// TIA Portal V20 export
FUNCTION_BLOCK "LER_Heater"   // FB21, LAD
// stored: Access Published, MemoryReserve 100, SetENOAutomatically false
   VAR_INPUT
      enable { ExternalAccessible := 'False'; ExternalVisible := 'False'; ExternalWritable := 'False'} : Bool;   // TRUE: Enable functionality of FB
      enableManualCmds : Bool;   // Enabling manual commands
      Clock : Bool;
   END_VAR
   VAR_OUTPUT
      Error : Bool;
   END_VAR
   VAR_IN_OUT
      ModbusMasterDataPTR : Variant;
      configuration : "LER_typeHeaterConfiguration";
      controlNode : "LER_typeHeaterControlNode";
      moduleInterface : "LER_typeHeaterInterface";
   END_VAR
   VAR
      statEnable : Bool;
      statEnableManualCmds : Bool;
      statSaveBtn : Bool;
      staSaveOneCycleDONE : Bool;
      instModbusCommLoad : Modbus_Comm_Load;
      instModbusMaster : Modbus_Master;
      instLER_Heater : Array[1.."Number_Of_E5CC"] of "LER_E5CC";
      "statE5CC[1]" { S7_SetPoint := 'True'} : "LER_typeE5CCStatus";
      "statE5CC[2]" { S7_SetPoint := 'True'} : "LER_typeE5CCStatus";
      "statE5CC[3]" { S7_SetPoint := 'True'} : "LER_typeE5CCStatus";
      "statE5CC[4]" { S7_SetPoint := 'True'} : "LER_typeE5CCStatus";
      "statE5CC[5]" { S7_SetPoint := 'True'} : "LER_typeE5CCStatus";
      statMBMasterBuffer { S7_SetPoint := 'True'} : Array[1.."Number_Of_E5CC"] of "LER_typeHeaterConfiguration_MB_Master";
      statCommand : "LER_typeHeaterCommands";
      statCMDKeep : Struct
         "E5CC[1]" : Struct
            Upper_Heater_Run : Bool;
            Upper_Heater_Stop : Bool;
            Upper_AutoTune_Run : Bool;
            Upper_AutoTune_Stop : Bool;
         END_STRUCT;
         "E5CC[2]" : Struct
            Upper_Heater_Run : Bool;
            Upper_Heater_Stop : Bool;
            Upper_AutoTune_Run : Bool;
            Upper_AutoTune_Stop : Bool;
         END_STRUCT;
         "E5CC[3]" : Struct
            Upper_Heater_Run : Bool;
            Upper_Heater_Stop : Bool;
            Upper_AutoTune_Run : Bool;
            Upper_AutoTune_Stop : Bool;
         END_STRUCT;
         "E5CC[4]" : Struct
            Upper_Heater_Run : Bool;
            Upper_Heater_Stop : Bool;
            Upper_AutoTune_Run : Bool;
            Upper_AutoTune_Stop : Bool;
         END_STRUCT;
         "E5CC[5]" : Struct
            Upper_Heater_Run : Bool;
            Upper_Heater_Stop : Bool;
            Upper_AutoTune_Run : Bool;
            Upper_AutoTune_Stop : Bool;
         END_STRUCT;
         E5CC1ReadStop : Bool;
         E5CC2ReadStop : Bool;
         E5CC3ReadStop : Bool;
         E5CC4ReadStop : Bool;
         E5CC5ReadStop : Bool;
      END_STRUCT;
      statConfiguration : "LER_typeHeaterConfiguration";
      statMonitoring { S7_SetPoint := 'True'} : "LER_typeHeaterMonitoring";
      statCurrentUnit : Int := 1;
      statTimer : Array[0..30] of TON_TIME;
      statPulse : Array[0..59] of Bool;
      IEC_Timer_0_Instance { S7_SetPoint := 'True'} : TOF_TIME;
      IEC_Timer_0_Instance_1 { S7_SetPoint := 'True'} : TOF_TIME;
      IEC_Timer_0_Instance_2 { S7_SetPoint := 'True'} : TOF_TIME;
      IEC_Timer_0_Instance_3 { S7_SetPoint := 'True'} : TOF_TIME;
      IEC_Timer_0_Instance_4 { S7_SetPoint := 'True'} : TOF_TIME;
   END_VAR
   VAR_TEMP
      tempErrInt : Int;
      tempErrWord : Word;
   END_VAR
   VAR CONSTANT
      Addr_TempPV : UDInt := 40001;
      Addr_Status : UDInt := 40003;
      Addr_TempSP : UDInt := 40263;
      Addr_AlarmValue1 : UDInt := 40265;
      Addr_AlarmValue1_UpperLimit : UDInt := 40267;
      Addr_AlarmValue1_LowerLimit : UDInt := 40269;
      Addr_AlarmValue2 : UDInt := 40271;
      Addr_AlarmValue2_UpperLimit : UDInt := 40273;
      Addr_AlarmValue2_LowerLimit : UDInt := 40275;
      CMD_Run : DWord := 16#01000000;
      CMD_Stop : DWord := 16#01010000;
      CMD_AutoTune_Run : DWord := 16#03020000;
      CMD_AutoTune_Stop : DWord := 16#03000000;
      Mode_Read : Int := 0;
      Mode_Write : Int := 1;
      Read_Time : Time := T#500MS;
      STATUS_NO_ERROR_OCCURRED : DWord;   // No error occurred.
      ERR_HEATER_CURRENT_VALUE_EXCEEDED_CT1 : DWord := 16#1;
      ERR_HEATER_CURRENT_VALUE_HOLD_CT1 : DWord := 16#2;
      ERR_AD_CONVERTER_ABNORMALITY : DWord := 16#4;
      ERR_HS_SSR_FAULT_ALERT_CT1 : DWord := 16#8;
      ERR_RSP_INPUT_ABNORMALITIES : DWord := 16#10;
      ERR_MORE_THAN_INPUT : DWord := 16#40;
      ERR_POTENTIOMETER_INPUT_ABNORMAL : DWord := 16#80;
      ERR_CONTROL_OUTPUT_HEATED_OPEN_OUTPUT : DWord := 16#100;
      ERR_CONTROL_OUTPUT_COOL_CLOSE_OUTPUT : DWord := 16#200;
      ERR_HEATER_OPEN_CIRCUIT_HB_ALARM_CT1 : DWord := 16#400;
      ERR_HEATER_OPEN_CIRCUIT_HB_ALARM_CT2 : DWord := 16#800;
      ERR_ALERT_1 : DWord := 16#1000;
      ERR_ALERT_2 : DWord := 16#2000;
      ERR_ALERT_3 : DWord := 16#4000;
      ERR_PROGRAM_END_OUTPUT : DWord := 16#8000;
      ERR_EVENT_INPUT_1 : DWord := 16#10000;
      ERR_EVENT_INPUT_2 : DWord := 16#20000;
      ERR_EVENT_INPUT_3 : DWord := 16#40000;
      ERR_EVENT_INPUT_4 : DWord := 16#80000;
      ERR_WRITE_MODE : DWord := 16#100000;
      ERR_NON_VOLATILE_MEMORY : DWord := 16#200000;
      ERR_SETTING_AREA : DWord := 16#400000;
      ERR_AT_RUN_STOP : DWord := 16#800000;
      ERR_RUN_STOP : DWord := 16#1000000;
      ERR_COMMUNICATION_WRITE : DWord := 16#2000000;
      ERR_AUTO_MANUAL : DWord := 16#4000000;
      ERR_PROGRAM_START : DWord := 16#8000000;
      ERR_HEATER_CURRENT_VALUE_EXCEEDED_CT2 : DWord := 16#10000000;
      ERR_HEATER_CURRENT_VALUE_HOLD_CT2 : DWord := 16#20000000;
      ERR_HS_SSR_FAILURE_ALARM_CT2 : DWord := 16#80000000;
   END_VAR
   VAR_TEMP   // added for the SCL form of the ladder/FBD networks
      _w1 : Bool;
      _w2 : Bool;
   END_VAR
BEGIN

REGION Network 1 (SCL): ###### Input Mapping ######
   // Main Common
   #statEnable := #enable;
   #statEnableManualCmds := #enableManualCmds;

   // Manual Command
   IF #statEnableManualCmds THEN
       #statCommand.Communication_Reset := #moduleInterface.commands.Communication_Reset;
       #statCommand.Save := #moduleInterface.commands.Save;
       #statCommand.Error_Reset := #moduleInterface.commands.Error_Reset;
       #statCommand.Upper_Heater_Run := #moduleInterface.commands.Upper_Heater_Run;
       #statCommand.Upper_Heater_Stop := #moduleInterface.commands.Upper_Heater_Stop;
       #statCommand.Upper_AutoTune_Run := #moduleInterface.commands.Upper_AutoTune_Run;
       #statCommand.Upper_AutoTune_Stop := #moduleInterface.commands.Upper_AutoTune_Stop;
       #statCommand.Lower_Heater_Run := #moduleInterface.commands.Lower_Heater_Run;
       #statCommand.Lower_Heater_Stop := #moduleInterface.commands.Lower_Heater_Stop;
       #statCommand.Lower_AutoTune_Run := #moduleInterface.commands.Lower_AutoTune_Run;
       #statCommand.Lower_AutoTune_Stop := #moduleInterface.commands.Lower_AutoTune_Stop;
       #statCommand.E5CC[1] := #moduleInterface.commands.E5CC[1];
       #statCommand.E5CC[2] := #moduleInterface.commands.E5CC[2];
       #statCommand.E5CC[3] := #moduleInterface.commands.E5CC[3];
       #statCommand.E5CC[4] := #moduleInterface.commands.E5CC[4];
       #statCommand.E5CC[5] := #moduleInterface.commands.E5CC[5];
   END_IF;

   // E5CC Config Setting
   IF #statCommand.Save OR #statCommand.Upper_Heater_Run THEN
       #statConfiguration.E5CC[1] := #moduleInterface.configuration.E5CC[1];
       #statConfiguration.E5CC[2] := #moduleInterface.configuration.E5CC[2];
       #statConfiguration.E5CC[3] := #moduleInterface.configuration.E5CC[3];
       #statConfiguration.E5CC[4] := #moduleInterface.configuration.E5CC[4];
       #statConfiguration.E5CC[5] := #moduleInterface.configuration.E5CC[5];
   END_IF;

   // 통신 에러시 자동 초기화
   IF NOT #statConfiguration.MB_Comm_Load.DONE THEN
       #statConfiguration.MB_Comm_Load.REQ := #Clock;
   ELSE
       #statConfiguration.MB_Comm_Load.REQ := FALSE;
   END_IF;

   // Modbus Comm Load Setting
   #statConfiguration.MB_Comm_Load.PORT := #configuration.MB_Comm_Load.PORT;
   #statConfiguration.MB_Comm_Load.BAUD := #configuration.MB_Comm_Load.BAUD;
   #statConfiguration.MB_Comm_Load.MB_DB := #instModbusMaster.MB_DB;
   #statConfiguration.MB_Comm_Load.PARITY := #configuration.MB_Comm_Load.PARITY;
   #instModbusCommLoad.MODE := 4; // **************** 매우 중요 ******************

   //Read Step Initialization
   IF #statCurrentUnit = 0 THEN
       #statCurrentUnit := 1;
   ELSIF #statCurrentUnit > "Number_Of_E5CC" THEN
       #statCurrentUnit := 1;
   END_IF;
END_REGION

REGION Network 2 (SCL): statCurrentUnit Mapping
   IF #statCurrentUnit = 1 THEN
       #statMBMasterBuffer[1].DONE := #statConfiguration.MB_Master.DONE;
       #statConfiguration.MB_Master.REQ := #statMBMasterBuffer[1].REQ;
       #statConfiguration.MB_Master.MB_ADDR := #statMBMasterBuffer[1].MB_ADDR;
       #statConfiguration.MB_Master.MODE := #statMBMasterBuffer[1].MODE;
       #statConfiguration.MB_Master.DATA_ADDR := #statMBMasterBuffer[1].DATA_ADDR;
       #statConfiguration.MB_Master.DATA_LEN := #statMBMasterBuffer[1].DATA_LEN;
       IF #statConfiguration.MB_Master.MODE = 0 THEN
           #tempErrInt := MOVE_BLK_VARIANT(SRC := #ModbusMasterDataPTR, COUNT := 20, SRC_INDEX := 0, DEST_INDEX := 0, DEST => #statMBMasterBuffer[1].DataPTR);
           #tempErrWord := INT_TO_WORD(IN := #tempErrInt);
       ELSIF #statConfiguration.MB_Master.MODE = 1 THEN
           #tempErrInt := MOVE_BLK_VARIANT(SRC := #statMBMasterBuffer[1].DataPTR, COUNT := 20, SRC_INDEX := 0, DEST_INDEX := 0, DEST => #ModbusMasterDataPTR);
           #tempErrWord := INT_TO_WORD(IN := #tempErrInt);
       END_IF;
   ELSE
       #statMBMasterBuffer[1].DONE := FALSE;
       #statMBMasterBuffer[1].REQ := FALSE;
       #statMBMasterBuffer[1].MB_ADDR := 0;
       #statMBMasterBuffer[1].MODE:= 0;
       #statMBMasterBuffer[1].DATA_ADDR := 0;
       #statMBMasterBuffer[1].DATA_LEN:= 0;
   END_IF;
   IF #statCurrentUnit = 2 THEN
       #statMBMasterBuffer[2].DONE := #statConfiguration.MB_Master.DONE;
       #statConfiguration.MB_Master.REQ := #statMBMasterBuffer[2].REQ;
       #statConfiguration.MB_Master.MB_ADDR := #statMBMasterBuffer[2].MB_ADDR;
       #statConfiguration.MB_Master.MODE := #statMBMasterBuffer[2].MODE;
       #statConfiguration.MB_Master.DATA_ADDR := #statMBMasterBuffer[2].DATA_ADDR;
       #statConfiguration.MB_Master.DATA_LEN := #statMBMasterBuffer[2].DATA_LEN;
       IF #statConfiguration.MB_Master.MODE = 0 THEN
           #tempErrInt := MOVE_BLK_VARIANT(SRC := #ModbusMasterDataPTR, COUNT := 20, SRC_INDEX := 0, DEST_INDEX := 0, DEST => #statMBMasterBuffer[2].DataPTR);
           #tempErrWord := INT_TO_WORD(IN := #tempErrInt);
       ELSIF #statConfiguration.MB_Master.MODE = 1 THEN
           #tempErrInt := MOVE_BLK_VARIANT(SRC := #statMBMasterBuffer[2].DataPTR, COUNT := 20, SRC_INDEX := 0, DEST_INDEX := 0, DEST => #ModbusMasterDataPTR);
           #tempErrWord := INT_TO_WORD(IN := #tempErrInt);
       END_IF;
   ELSE
       #statMBMasterBuffer[2].DONE := FALSE;
       #statMBMasterBuffer[2].REQ := FALSE;
       #statMBMasterBuffer[2].MB_ADDR := 0;
       #statMBMasterBuffer[2].MODE := 0;
       #statMBMasterBuffer[2].DATA_ADDR := 0;
       #statMBMasterBuffer[2].DATA_LEN := 0;
   END_IF;
   IF #statCurrentUnit = 3 THEN
       #statMBMasterBuffer[3].DONE := #statConfiguration.MB_Master.DONE;
       #statConfiguration.MB_Master.REQ := #statMBMasterBuffer[3].REQ;
       #statConfiguration.MB_Master.MB_ADDR := #statMBMasterBuffer[3].MB_ADDR;
       #statConfiguration.MB_Master.MODE := #statMBMasterBuffer[3].MODE;
       #statConfiguration.MB_Master.DATA_ADDR := #statMBMasterBuffer[3].DATA_ADDR;
       #statConfiguration.MB_Master.DATA_LEN := #statMBMasterBuffer[3].DATA_LEN;
       IF #statConfiguration.MB_Master.MODE = 0 THEN
           #tempErrInt := MOVE_BLK_VARIANT(SRC := #ModbusMasterDataPTR, COUNT := 20, SRC_INDEX := 0, DEST_INDEX := 0, DEST => #statMBMasterBuffer[3].DataPTR);
           #tempErrWord := INT_TO_WORD(IN := #tempErrInt);
       ELSIF #statConfiguration.MB_Master.MODE = 1 THEN
           #tempErrInt := MOVE_BLK_VARIANT(SRC := #statMBMasterBuffer[3].DataPTR, COUNT := 20, SRC_INDEX := 0, DEST_INDEX := 0, DEST => #ModbusMasterDataPTR);
           #tempErrWord := INT_TO_WORD(IN := #tempErrInt);
       END_IF;
   ELSE
       #statMBMasterBuffer[3].DONE := FALSE;
       #statMBMasterBuffer[3].REQ := FALSE;
       #statMBMasterBuffer[3].MB_ADDR := 0;
       #statMBMasterBuffer[3].MODE := 0;
       #statMBMasterBuffer[3].DATA_ADDR := 0;
       #statMBMasterBuffer[3].DATA_LEN := 0;
   END_IF;
   IF #statCurrentUnit = 4 THEN
       #statMBMasterBuffer[4].DONE := #statConfiguration.MB_Master.DONE;
       #statConfiguration.MB_Master.REQ := #statMBMasterBuffer[4].REQ;
       #statConfiguration.MB_Master.MB_ADDR := #statMBMasterBuffer[4].MB_ADDR;
       #statConfiguration.MB_Master.MODE := #statMBMasterBuffer[4].MODE;
       #statConfiguration.MB_Master.DATA_ADDR := #statMBMasterBuffer[4].DATA_ADDR;
       #statConfiguration.MB_Master.DATA_LEN := #statMBMasterBuffer[4].DATA_LEN;
       IF #statConfiguration.MB_Master.MODE = 0 THEN
           #tempErrInt := MOVE_BLK_VARIANT(SRC := #ModbusMasterDataPTR, COUNT := 20, SRC_INDEX := 0, DEST_INDEX := 0, DEST => #statMBMasterBuffer[4].DataPTR);
           #tempErrWord := INT_TO_WORD(IN := #tempErrInt);
       ELSIF #statConfiguration.MB_Master.MODE = 1 THEN
           #tempErrInt := MOVE_BLK_VARIANT(SRC := #statMBMasterBuffer[4].DataPTR, COUNT := 20, SRC_INDEX := 0, DEST_INDEX := 0, DEST => #ModbusMasterDataPTR);
           #tempErrWord := INT_TO_WORD(IN := #tempErrInt);
       END_IF;
   ELSE
       #statMBMasterBuffer[4].DONE := FALSE;
       #statMBMasterBuffer[4].REQ := FALSE;
       #statMBMasterBuffer[4].MB_ADDR := 0;
       #statMBMasterBuffer[4].MODE := 0;
       #statMBMasterBuffer[4].DATA_ADDR := 0;
       #statMBMasterBuffer[4].DATA_LEN := 0;
   END_IF;
   IF #statCurrentUnit = 5 THEN
       #statMBMasterBuffer[5].DONE := #statConfiguration.MB_Master.DONE;
       #statConfiguration.MB_Master.REQ := #statMBMasterBuffer[5].REQ;
       #statConfiguration.MB_Master.MB_ADDR := #statMBMasterBuffer[5].MB_ADDR;
       #statConfiguration.MB_Master.MODE := #statMBMasterBuffer[5].MODE;
       #statConfiguration.MB_Master.DATA_ADDR := #statMBMasterBuffer[5].DATA_ADDR;
       #statConfiguration.MB_Master.DATA_LEN := #statMBMasterBuffer[5].DATA_LEN;
       IF #statConfiguration.MB_Master.MODE = 0 THEN
           #tempErrInt := MOVE_BLK_VARIANT(SRC := #ModbusMasterDataPTR, COUNT := 20, SRC_INDEX := 0, DEST_INDEX := 0, DEST => #statMBMasterBuffer[5].DataPTR);
           #tempErrWord := INT_TO_WORD(IN := #tempErrInt);
       ELSIF #statConfiguration.MB_Master.MODE = 1 THEN
           #tempErrInt := MOVE_BLK_VARIANT(SRC := #statMBMasterBuffer[5].DataPTR, COUNT := 20, SRC_INDEX := 0, DEST_INDEX := 0, DEST => #ModbusMasterDataPTR);
           #tempErrWord := INT_TO_WORD(IN := #tempErrInt);
       END_IF;
   ELSE
       #statMBMasterBuffer[5].DONE := FALSE;
       #statMBMasterBuffer[5].REQ := FALSE;
       #statMBMasterBuffer[5].MB_ADDR := 0;
       #statMBMasterBuffer[5].MODE := 0;
       #statMBMasterBuffer[5].DATA_ADDR := 0;
       #statMBMasterBuffer[5].DATA_LEN := 0;
   END_IF;
END_REGION

REGION Network 3: Commoon Error Reset
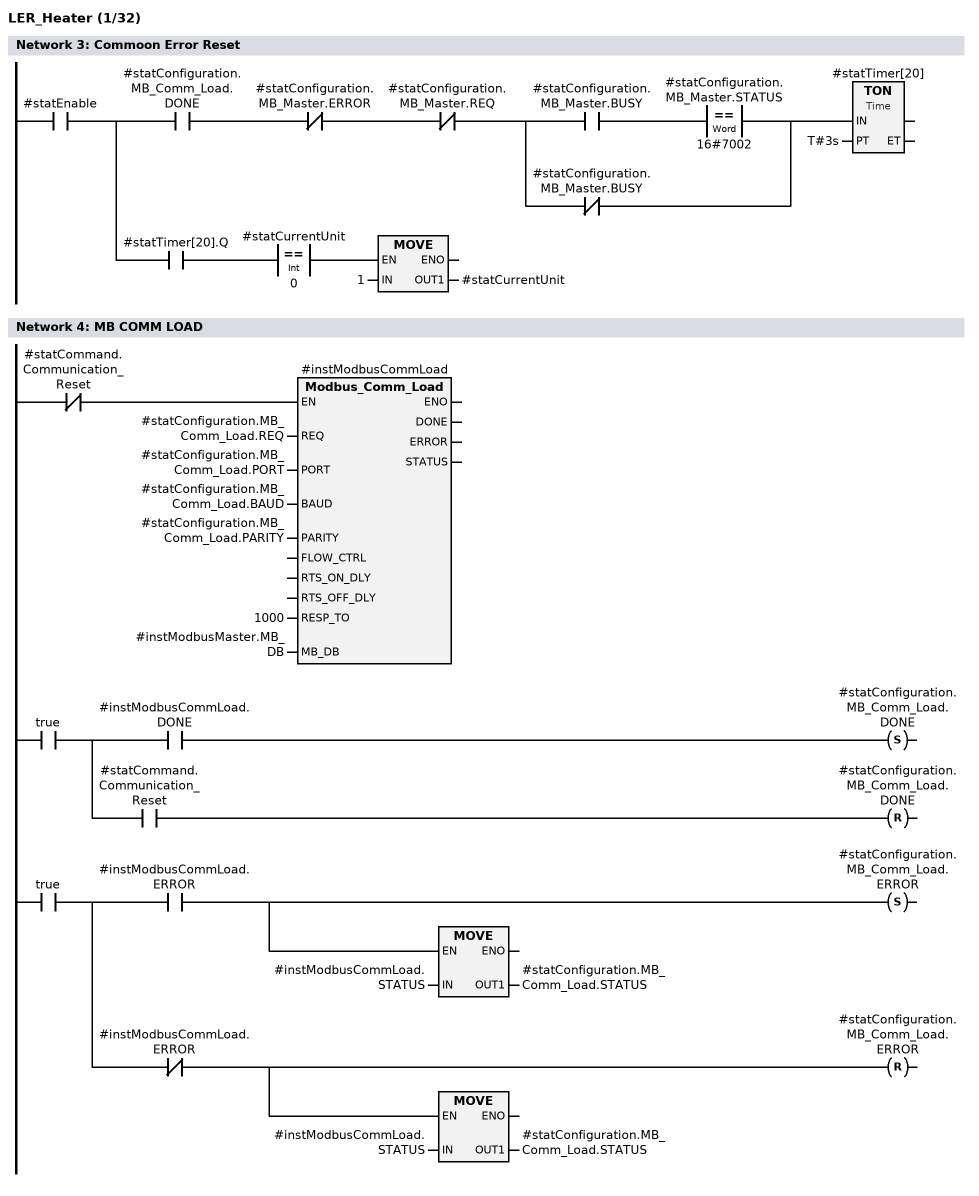
   RUNG wire#powerrail
      Contact( #statEnable )
      wire#w1
      Contact( #statConfiguration.MB_Comm_Load.DONE )
      I_Contact( #statConfiguration.MB_Master.ERROR )
      I_Contact( #statConfiguration.MB_Master.REQ )
      wire#w2
      Contact( #statConfiguration.MB_Master.BUSY )
      { S7_Templates := "SrcType := Word" } EQ_Contact(in1 := #statConfiguration.MB_Master.STATUS, in2 := 16#7002)
      wire#w3
      { S7_Templates := "time_type := Time" } #statTimer[20].TON(pt := T#3s, et =>)
   END_RUNG
   RUNG wire#w2
      I_Contact( #statConfiguration.MB_Master.BUSY )
   END_RUNG wire#w3
   RUNG wire#w1
      Contact( #statTimer[20].Q )
      { S7_Templates := "SrcType := Int" } EQ_Contact(in1 := #statCurrentUnit, in2 := 0)
      Move(in := 1, out1 => #statCurrentUnit)
   END_RUNG
   // the same network as SCL:
   #statTimer[20].TON(IN := #statEnable AND #statConfiguration.MB_Comm_Load.DONE AND NOT #statConfiguration.MB_Master.ERROR AND NOT #statConfiguration.MB_Master.REQ AND ((#statConfiguration.MB_Master.BUSY AND (#statConfiguration.MB_Master.STATUS = 16#7002)) OR NOT #statConfiguration.MB_Master.BUSY),
                      PT := T#3s);
   IF #statEnable AND #statTimer[20].Q AND (#statCurrentUnit = 0) THEN #statCurrentUnit := 1; END_IF;
END_REGION

REGION Network 4: MB COMM LOAD
   RUNG wire#powerrail
      I_Contact( #statCommand.Communication_Reset )
      #instModbusCommLoad.Modbus_Comm_Load(REQ := #statConfiguration.MB_Comm_Load.REQ, PORT := #statConfiguration.MB_Comm_Load.PORT, BAUD := #statConfiguration.MB_Comm_Load.BAUD, PARITY := #statConfiguration.MB_Comm_Load.PARITY, FLOW_CTRL :=, RTS_ON_DLY :=, RTS_OFF_DLY :=, RESP_TO := 1000, MB_DB := #instModbusMaster.MB_DB, DONE =>, ERROR =>, STATUS =>)
   END_RUNG
   RUNG wire#powerrail
      Contact( true )
      wire#w1
      Contact( #instModbusCommLoad.DONE )
      S_Coil( #statConfiguration.MB_Comm_Load.DONE )
   END_RUNG
   RUNG wire#w1
      Contact( #statCommand.Communication_Reset )
      R_Coil( #statConfiguration.MB_Comm_Load.DONE )
   END_RUNG
   RUNG wire#powerrail
      Contact( true )
      wire#w2
      Contact( #instModbusCommLoad.ERROR )
      wire#w3
      S_Coil( #statConfiguration.MB_Comm_Load.ERROR )
   END_RUNG
   RUNG wire#w3
      Move(in := #instModbusCommLoad.STATUS, out1 => #statConfiguration.MB_Comm_Load.STATUS)
   END_RUNG
   RUNG wire#w2
      I_Contact( #instModbusCommLoad.ERROR )
      wire#w4
      R_Coil( #statConfiguration.MB_Comm_Load.ERROR )
   END_RUNG
   RUNG wire#w4
      Move(in := #instModbusCommLoad.STATUS, out1 => #statConfiguration.MB_Comm_Load.STATUS)
   END_RUNG
   // the same network as SCL:
   IF NOT #statCommand.Communication_Reset THEN
       #instModbusCommLoad(REQ := #statConfiguration.MB_Comm_Load.REQ,   // Modbus_Comm_Load
                           PORT := #statConfiguration.MB_Comm_Load.PORT,
                           BAUD := #statConfiguration.MB_Comm_Load.BAUD,
                           PARITY := #statConfiguration.MB_Comm_Load.PARITY,
                           RESP_TO := 1000,
                           MB_DB := #instModbusMaster.MB_DB);
   END_IF;
   IF true AND #instModbusCommLoad.DONE THEN #statConfiguration.MB_Comm_Load.DONE := TRUE; END_IF;
   IF true AND #statCommand.Communication_Reset THEN #statConfiguration.MB_Comm_Load.DONE := FALSE; END_IF;
   IF true AND #instModbusCommLoad.ERROR THEN
       #statConfiguration.MB_Comm_Load.ERROR := TRUE;
       #statConfiguration.MB_Comm_Load.STATUS := #instModbusCommLoad.STATUS;
   END_IF;
   IF true AND NOT #instModbusCommLoad.ERROR THEN
       #statConfiguration.MB_Comm_Load.ERROR := FALSE;
       #statConfiguration.MB_Comm_Load.STATUS := #instModbusCommLoad.STATUS;
   END_IF;
END_REGION

REGION Network 5: MB MASTER
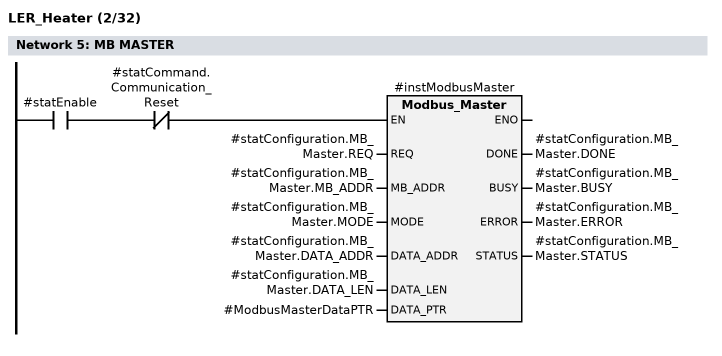
   RUNG wire#powerrail
      Contact( #statEnable )
      I_Contact( #statCommand.Communication_Reset )
      #instModbusMaster.Modbus_Master(REQ := #statConfiguration.MB_Master.REQ, MB_ADDR := #statConfiguration.MB_Master.MB_ADDR, MODE := #statConfiguration.MB_Master.MODE, DATA_ADDR := #statConfiguration.MB_Master.DATA_ADDR, DATA_LEN := #statConfiguration.MB_Master.DATA_LEN, DATA_PTR := #ModbusMasterDataPTR, DONE => #statConfiguration.MB_Master.DONE, BUSY => #statConfiguration.MB_Master.BUSY, ERROR => #statConfiguration.MB_Master.ERROR, STATUS => #statConfiguration.MB_Master.STATUS)
   END_RUNG
   // the same network as SCL:
   IF #statEnable AND NOT #statCommand.Communication_Reset THEN
       #instModbusMaster(REQ := #statConfiguration.MB_Master.REQ,   // Modbus_Master
                         MB_ADDR := #statConfiguration.MB_Master.MB_ADDR,
                         MODE := #statConfiguration.MB_Master.MODE,
                         DATA_ADDR := #statConfiguration.MB_Master.DATA_ADDR,
                         DATA_LEN := #statConfiguration.MB_Master.DATA_LEN,
                         DATA_PTR := #ModbusMasterDataPTR,
                         DONE => #statConfiguration.MB_Master.DONE,
                         BUSY => #statConfiguration.MB_Master.BUSY,
                         ERROR => #statConfiguration.MB_Master.ERROR,
                         STATUS => #statConfiguration.MB_Master.STATUS);
   END_IF;
END_REGION

REGION Network 6: E5CC[1] - ###### Input Mapping ######
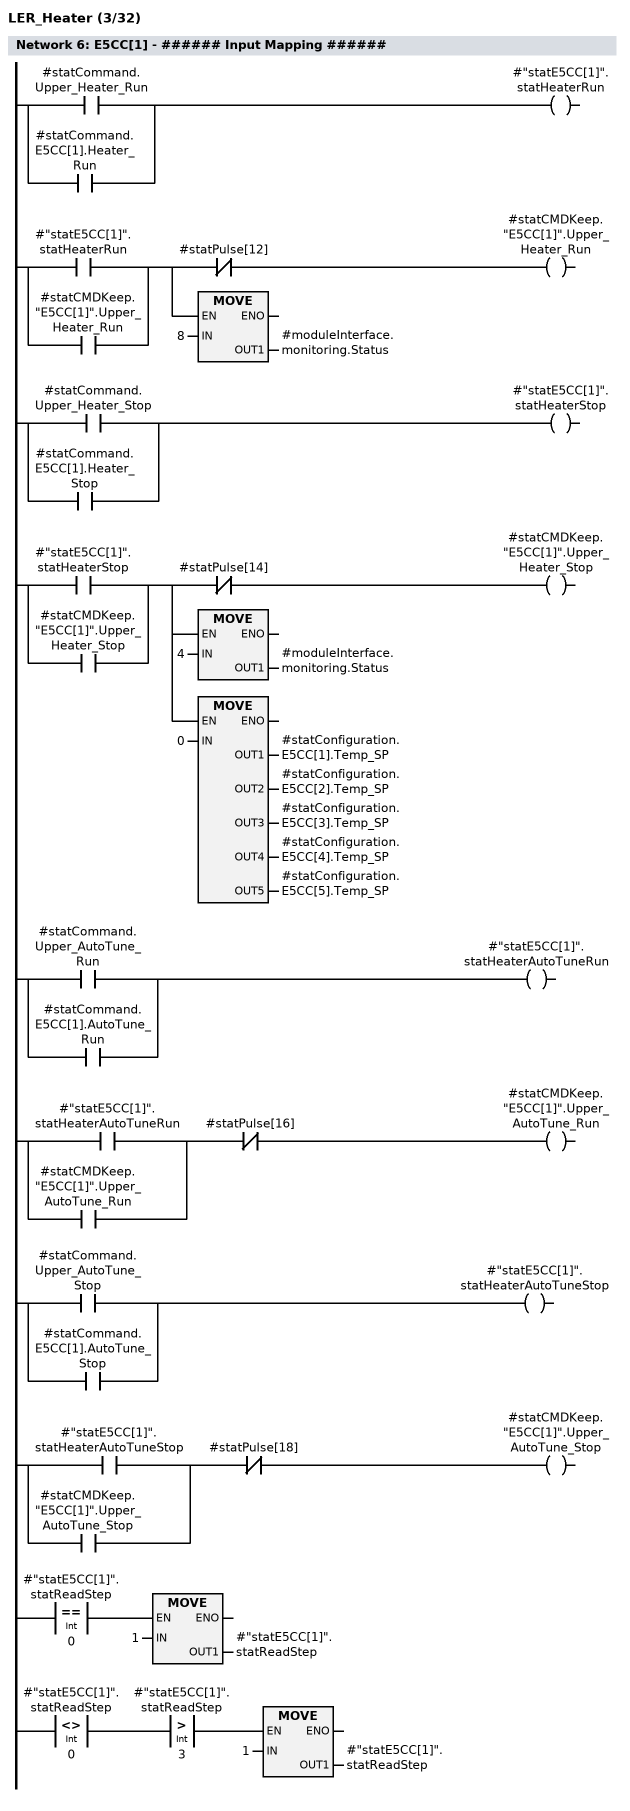
   RUNG wire#powerrail
      Contact( #statCommand.Upper_Heater_Run )
      wire#w1
      Coil( #"statE5CC[1]".statHeaterRun )
   END_RUNG
   RUNG wire#powerrail
      Contact( #statCommand.E5CC[1].Heater_Run )
   END_RUNG wire#w1
   RUNG wire#powerrail
      Contact( #"statE5CC[1]".statHeaterRun )
      wire#w2
      I_Contact( #statPulse[12] )
      Coil( #statCMDKeep."E5CC[1]".Upper_Heater_Run )
   END_RUNG
   RUNG wire#powerrail
      Contact( #statCMDKeep."E5CC[1]".Upper_Heater_Run )
   END_RUNG wire#w2
   RUNG wire#w2
      Move(in := 8, out1 => #moduleInterface.monitoring.Status)
   END_RUNG
   RUNG wire#powerrail
      Contact( #statCommand.Upper_Heater_Stop )
      wire#w3
      Coil( #"statE5CC[1]".statHeaterStop )
   END_RUNG
   RUNG wire#powerrail
      Contact( #statCommand.E5CC[1].Heater_Stop )
   END_RUNG wire#w3
   RUNG wire#powerrail
      Contact( #"statE5CC[1]".statHeaterStop )
      wire#w4
      I_Contact( #statPulse[14] )
      Coil( #statCMDKeep."E5CC[1]".Upper_Heater_Stop )
   END_RUNG
   RUNG wire#powerrail
      Contact( #statCMDKeep."E5CC[1]".Upper_Heater_Stop )
   END_RUNG wire#w4
   RUNG wire#w4
      Move(in := 4, out1 => #moduleInterface.monitoring.Status)
   END_RUNG
   RUNG wire#w4
      Move(in := 0, out1 => #statConfiguration.E5CC[1].Temp_SP, out2 => #statConfiguration.E5CC[2].Temp_SP, out3 => #statConfiguration.E5CC[3].Temp_SP, out4 => #statConfiguration.E5CC[4].Temp_SP, out5 => #statConfiguration.E5CC[5].Temp_SP)
   END_RUNG
   RUNG wire#powerrail
      Contact( #statCommand.Upper_AutoTune_Run )
      wire#w5
      Coil( #"statE5CC[1]".statHeaterAutoTuneRun )
   END_RUNG
   RUNG wire#powerrail
      Contact( #statCommand.E5CC[1].AutoTune_Run )
   END_RUNG wire#w5
   RUNG wire#powerrail
      Contact( #"statE5CC[1]".statHeaterAutoTuneRun )
      wire#w6
      I_Contact( #statPulse[16] )
      Coil( #statCMDKeep."E5CC[1]".Upper_AutoTune_Run )
   END_RUNG
   RUNG wire#powerrail
      Contact( #statCMDKeep."E5CC[1]".Upper_AutoTune_Run )
   END_RUNG wire#w6
   RUNG wire#powerrail
      Contact( #statCommand.Upper_AutoTune_Stop )
      wire#w7
      Coil( #"statE5CC[1]".statHeaterAutoTuneStop )
   END_RUNG
   RUNG wire#powerrail
      Contact( #statCommand.E5CC[1].AutoTune_Stop )
   END_RUNG wire#w7
   RUNG wire#powerrail
      Contact( #"statE5CC[1]".statHeaterAutoTuneStop )
      wire#w8
      I_Contact( #statPulse[18] )
      Coil( #statCMDKeep."E5CC[1]".Upper_AutoTune_Stop )
   END_RUNG
   RUNG wire#powerrail
      Contact( #statCMDKeep."E5CC[1]".Upper_AutoTune_Stop )
   END_RUNG wire#w8
   RUNG wire#powerrail
      { S7_Templates := "SrcType := Int" } EQ_Contact(in1 := #"statE5CC[1]".statReadStep, in2 := 0)
      Move(in := 1, out1 => #"statE5CC[1]".statReadStep)
   END_RUNG
   RUNG wire#powerrail
      { S7_Templates := "SrcType := Int" } NE_Contact(in1 := #"statE5CC[1]".statReadStep, in2 := 0)
      { S7_Templates := "SrcType := Int" } GT_Contact(in1 := #"statE5CC[1]".statReadStep, in2 := 3)
      Move(in := 1, out1 => #"statE5CC[1]".statReadStep)
   END_RUNG
   // the same network as SCL:
   #"statE5CC[1]".statHeaterRun := #statCommand.Upper_Heater_Run OR #statCommand.E5CC[1].Heater_Run;
   #_w1 := #"statE5CC[1]".statHeaterRun OR #statCMDKeep."E5CC[1]".Upper_Heater_Run;
   #statCMDKeep."E5CC[1]".Upper_Heater_Run := #_w1 AND NOT #statPulse[12];
   IF #_w1 THEN #moduleInterface.monitoring.Status := 8; END_IF;
   #"statE5CC[1]".statHeaterStop := #statCommand.Upper_Heater_Stop OR #statCommand.E5CC[1].Heater_Stop;
   #_w2 := #"statE5CC[1]".statHeaterStop OR #statCMDKeep."E5CC[1]".Upper_Heater_Stop;
   #statCMDKeep."E5CC[1]".Upper_Heater_Stop := #_w2 AND NOT #statPulse[14];
   IF #_w2 THEN
       #moduleInterface.monitoring.Status := 4;
       #statConfiguration.E5CC[1].Temp_SP := 0;
       #statConfiguration.E5CC[2].Temp_SP := 0;
       #statConfiguration.E5CC[3].Temp_SP := 0;
       #statConfiguration.E5CC[4].Temp_SP := 0;
       #statConfiguration.E5CC[5].Temp_SP := 0;
   END_IF;
   #"statE5CC[1]".statHeaterAutoTuneRun := #statCommand.Upper_AutoTune_Run OR #statCommand.E5CC[1].AutoTune_Run;
   #statCMDKeep."E5CC[1]".Upper_AutoTune_Run := (#"statE5CC[1]".statHeaterAutoTuneRun OR #statCMDKeep."E5CC[1]".Upper_AutoTune_Run) AND NOT #statPulse[16];
   #"statE5CC[1]".statHeaterAutoTuneStop := #statCommand.Upper_AutoTune_Stop OR #statCommand.E5CC[1].AutoTune_Stop;
   #statCMDKeep."E5CC[1]".Upper_AutoTune_Stop := (#"statE5CC[1]".statHeaterAutoTuneStop OR #statCMDKeep."E5CC[1]".Upper_AutoTune_Stop) AND NOT #statPulse[18];
   IF #"statE5CC[1]".statReadStep = 0 THEN #"statE5CC[1]".statReadStep := 1; END_IF;
   IF (#"statE5CC[1]".statReadStep <> 0) AND (#"statE5CC[1]".statReadStep > 3) THEN
       #"statE5CC[1]".statReadStep := 1;
   END_IF;
END_REGION

REGION Network 7: Read Condition
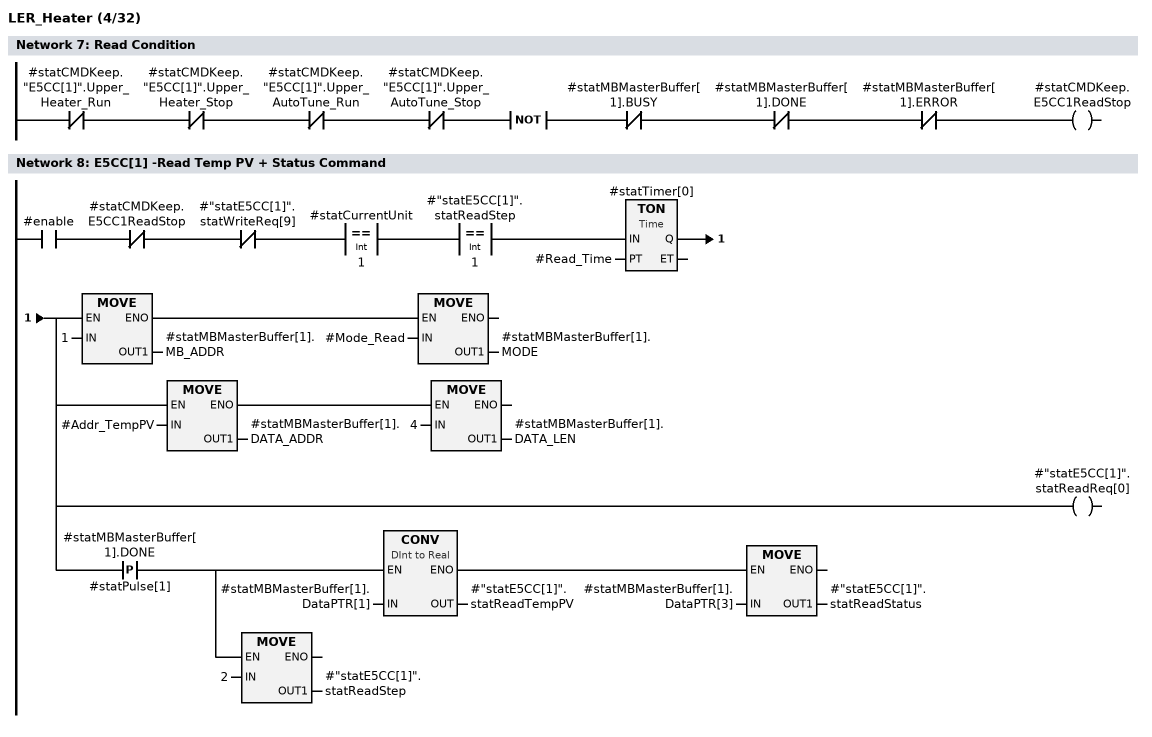
   RUNG wire#powerrail
      I_Contact( #statCMDKeep."E5CC[1]".Upper_Heater_Run )
      I_Contact( #statCMDKeep."E5CC[1]".Upper_Heater_Stop )
      I_Contact( #statCMDKeep."E5CC[1]".Upper_AutoTune_Run )
      I_Contact( #statCMDKeep."E5CC[1]".Upper_AutoTune_Stop )
      Not()
      I_Contact( #statMBMasterBuffer[1].BUSY )
      I_Contact( #statMBMasterBuffer[1].DONE )
      I_Contact( #statMBMasterBuffer[1].ERROR )
      Coil( #statCMDKeep.E5CC1ReadStop )
   END_RUNG
   // the same network as SCL:
   #statCMDKeep.E5CC1ReadStop := NOT (NOT #statCMDKeep."E5CC[1]".Upper_Heater_Run AND NOT #statCMDKeep."E5CC[1]".Upper_Heater_Stop AND NOT #statCMDKeep."E5CC[1]".Upper_AutoTune_Run AND NOT #statCMDKeep."E5CC[1]".Upper_AutoTune_Stop) AND NOT #statMBMasterBuffer[1].BUSY AND NOT #statMBMasterBuffer[1].DONE AND NOT #statMBMasterBuffer[1].ERROR;
END_REGION

REGION Network 8: E5CC[1] -Read Temp PV + Status Command
   RUNG wire#powerrail
      Contact( #enable )
      I_Contact( #statCMDKeep.E5CC1ReadStop )
      I_Contact( #"statE5CC[1]".statWriteReq[9] )
      { S7_Templates := "SrcType := Int" } EQ_Contact(in1 := #statCurrentUnit, in2 := 1)
      { S7_Templates := "SrcType := Int" } EQ_Contact(in1 := #"statE5CC[1]".statReadStep, in2 := 1)
      { S7_Templates := "time_type := Time" } #statTimer[0].TON(pt := #Read_Time, et =>)
      wire#w1
      Move(in := 1, out1 => #statMBMasterBuffer[1].MB_ADDR)
      Move(in := #Mode_Read, out1 => #statMBMasterBuffer[1].MODE)
   END_RUNG
   RUNG wire#w1
      Move(in := #Addr_TempPV, out1 => #statMBMasterBuffer[1].DATA_ADDR)
      Move(in := 4, out1 => #statMBMasterBuffer[1].DATA_LEN)
   END_RUNG
   RUNG wire#w1
      Coil( #"statE5CC[1]".statReadReq[0] )
   END_RUNG
   RUNG wire#w1
      P_Contact(operand := #statMBMasterBuffer[1].DONE, bit := #statPulse[1])
      wire#w2
      { S7_Templates := "[SrcType := DInt, DestType := Real]" } Convert(in := #statMBMasterBuffer[1].DataPTR[1], out => #"statE5CC[1]".statReadTempPV)
      Move(in := #statMBMasterBuffer[1].DataPTR[3], out1 => #"statE5CC[1]".statReadStatus)
   END_RUNG
   RUNG wire#w2
      Move(in := 2, out1 => #"statE5CC[1]".statReadStep)
   END_RUNG
   // the same network as SCL:
   #statTimer[0].TON(IN := #enable AND NOT #statCMDKeep.E5CC1ReadStop AND NOT #"statE5CC[1]".statWriteReq[9] AND (#statCurrentUnit = 1) AND (#"statE5CC[1]".statReadStep = 1),
                     PT := #Read_Time);
   IF #statTimer[0].Q THEN
       #statMBMasterBuffer[1].MB_ADDR := 1;
       #statMBMasterBuffer[1].MODE := #Mode_Read;
       #statMBMasterBuffer[1].DATA_ADDR := #Addr_TempPV;
       #statMBMasterBuffer[1].DATA_LEN := 4;
   END_IF;
   #"statE5CC[1]".statReadReq[0] := #statTimer[0].Q;
   #_w1 := #statTimer[0].Q AND #statMBMasterBuffer[1].DONE AND NOT #statPulse[1];   // rising edge of #statMBMasterBuffer[1].DONE
   #statPulse[1] := #statMBMasterBuffer[1].DONE;
   IF #_w1 THEN
       #"statE5CC[1]".statReadTempPV := DINT_TO_REAL(#statMBMasterBuffer[1].DataPTR[1]);
       #"statE5CC[1]".statReadStatus := #statMBMasterBuffer[1].DataPTR[3];
       #"statE5CC[1]".statReadStep := 2;
   END_IF;
END_REGION

REGION Network 9: E5CC[1] -Read TempSP + AlarmValue1 ~ AlarmValue2_LowerLimit Commad
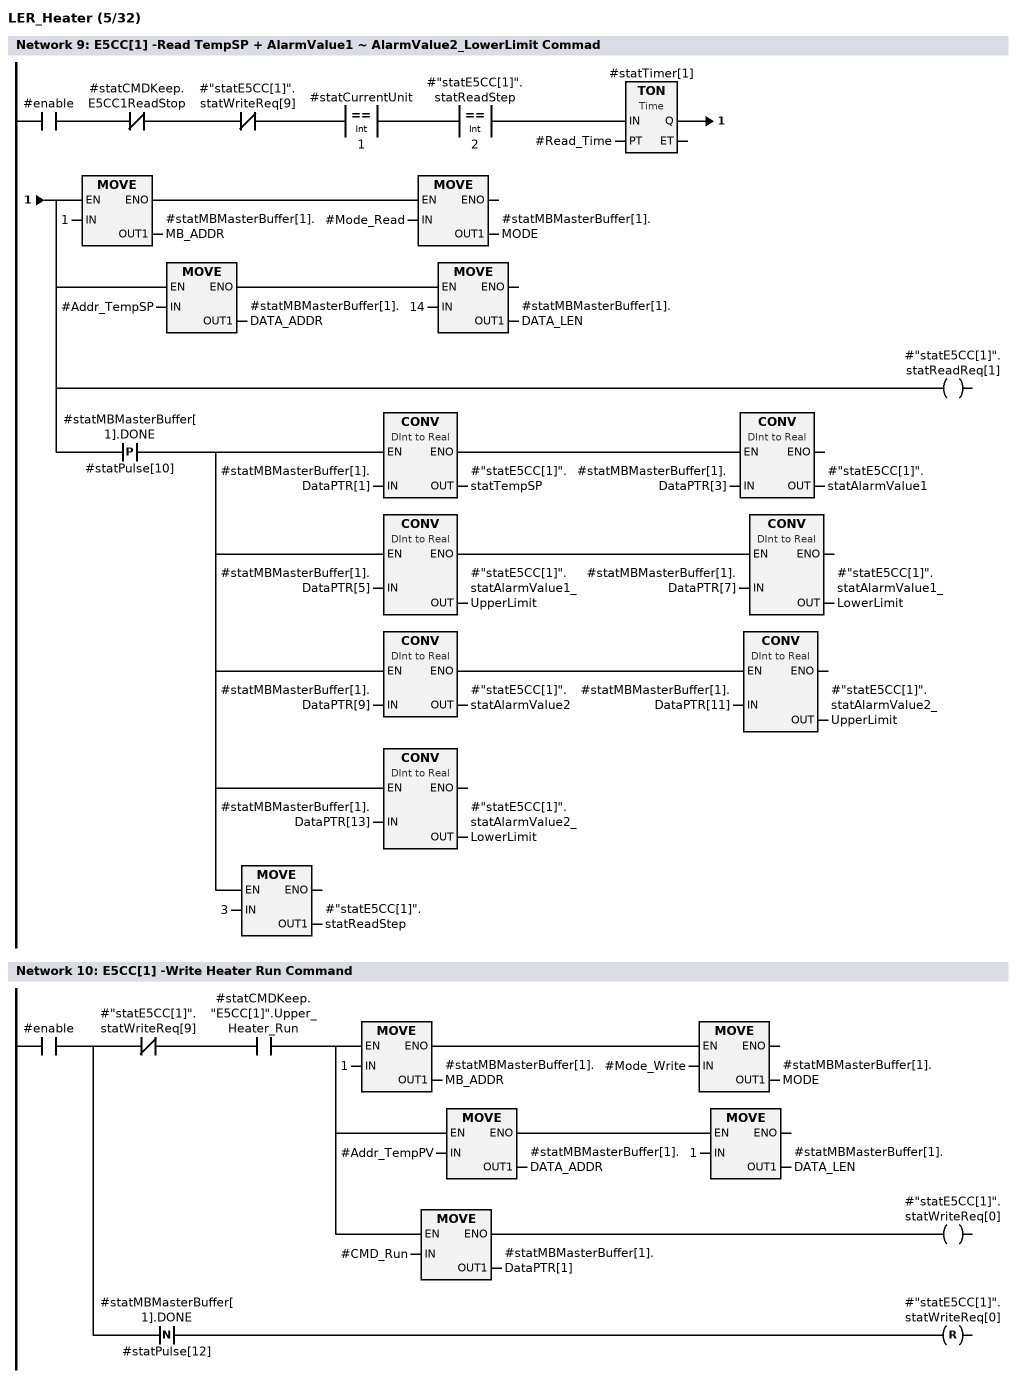
   RUNG wire#powerrail
      Contact( #enable )
      I_Contact( #statCMDKeep.E5CC1ReadStop )
      I_Contact( #"statE5CC[1]".statWriteReq[9] )
      { S7_Templates := "SrcType := Int" } EQ_Contact(in1 := #statCurrentUnit, in2 := 1)
      { S7_Templates := "SrcType := Int" } EQ_Contact(in1 := #"statE5CC[1]".statReadStep, in2 := 2)
      { S7_Templates := "time_type := Time" } #statTimer[1].TON(pt := #Read_Time, et =>)
      wire#w1
      Move(in := 1, out1 => #statMBMasterBuffer[1].MB_ADDR)
      Move(in := #Mode_Read, out1 => #statMBMasterBuffer[1].MODE)
   END_RUNG
   RUNG wire#w1
      Move(in := #Addr_TempSP, out1 => #statMBMasterBuffer[1].DATA_ADDR)
      Move(in := 14, out1 => #statMBMasterBuffer[1].DATA_LEN)
   END_RUNG
   RUNG wire#w1
      Coil( #"statE5CC[1]".statReadReq[1] )
   END_RUNG
   RUNG wire#w1
      P_Contact(operand := #statMBMasterBuffer[1].DONE, bit := #statPulse[10])
      wire#w2
      { S7_Templates := "[SrcType := DInt, DestType := Real]" } Convert(in := #statMBMasterBuffer[1].DataPTR[1], out => #"statE5CC[1]".statTempSP)
      { S7_Templates := "[SrcType := DInt, DestType := Real]" } Convert(in := #statMBMasterBuffer[1].DataPTR[3], out => #"statE5CC[1]".statAlarmValue1)
   END_RUNG
   RUNG wire#w2
      { S7_Templates := "[SrcType := DInt, DestType := Real]" } Convert(in := #statMBMasterBuffer[1].DataPTR[5], out => #"statE5CC[1]".statAlarmValue1_UpperLimit)
      { S7_Templates := "[SrcType := DInt, DestType := Real]" } Convert(in := #statMBMasterBuffer[1].DataPTR[7], out => #"statE5CC[1]".statAlarmValue1_LowerLimit)
   END_RUNG
   RUNG wire#w2
      { S7_Templates := "[SrcType := DInt, DestType := Real]" } Convert(in := #statMBMasterBuffer[1].DataPTR[9], out => #"statE5CC[1]".statAlarmValue2)
      { S7_Templates := "[SrcType := DInt, DestType := Real]" } Convert(in := #statMBMasterBuffer[1].DataPTR[11], out => #"statE5CC[1]".statAlarmValue2_UpperLimit)
   END_RUNG
   RUNG wire#w2
      { S7_Templates := "[SrcType := DInt, DestType := Real]" } Convert(in := #statMBMasterBuffer[1].DataPTR[13], out => #"statE5CC[1]".statAlarmValue2_LowerLimit)
   END_RUNG
   RUNG wire#w2
      Move(in := 3, out1 => #"statE5CC[1]".statReadStep)
   END_RUNG
   // the same network as SCL:
   #statTimer[1].TON(IN := #enable AND NOT #statCMDKeep.E5CC1ReadStop AND NOT #"statE5CC[1]".statWriteReq[9] AND (#statCurrentUnit = 1) AND (#"statE5CC[1]".statReadStep = 2),
                     PT := #Read_Time);
   IF #statTimer[1].Q THEN
       #statMBMasterBuffer[1].MB_ADDR := 1;
       #statMBMasterBuffer[1].MODE := #Mode_Read;
       #statMBMasterBuffer[1].DATA_ADDR := #Addr_TempSP;
       #statMBMasterBuffer[1].DATA_LEN := 14;
   END_IF;
   #"statE5CC[1]".statReadReq[1] := #statTimer[1].Q;
   #_w1 := #statTimer[1].Q AND #statMBMasterBuffer[1].DONE AND NOT #statPulse[10];   // rising edge of #statMBMasterBuffer[1].DONE
   #statPulse[10] := #statMBMasterBuffer[1].DONE;
   IF #_w1 THEN
       #"statE5CC[1]".statTempSP := DINT_TO_REAL(#statMBMasterBuffer[1].DataPTR[1]);
       #"statE5CC[1]".statAlarmValue1 := DINT_TO_REAL(#statMBMasterBuffer[1].DataPTR[3]);
       #"statE5CC[1]".statAlarmValue1_UpperLimit := DINT_TO_REAL(#statMBMasterBuffer[1].DataPTR[5]);
       #"statE5CC[1]".statAlarmValue1_LowerLimit := DINT_TO_REAL(#statMBMasterBuffer[1].DataPTR[7]);
       #"statE5CC[1]".statAlarmValue2 := DINT_TO_REAL(#statMBMasterBuffer[1].DataPTR[9]);
       #"statE5CC[1]".statAlarmValue2_UpperLimit := DINT_TO_REAL(#statMBMasterBuffer[1].DataPTR[11]);
       #"statE5CC[1]".statAlarmValue2_LowerLimit := DINT_TO_REAL(#statMBMasterBuffer[1].DataPTR[13]);
       #"statE5CC[1]".statReadStep := 3;
   END_IF;
END_REGION

REGION Network 10: E5CC[1] -Write Heater Run Command
   RUNG wire#powerrail
      Contact( #enable )
      wire#w1
      I_Contact( #"statE5CC[1]".statWriteReq[9] )
      Contact( #statCMDKeep."E5CC[1]".Upper_Heater_Run )
      wire#w2
      Move(in := 1, out1 => #statMBMasterBuffer[1].MB_ADDR)
      Move(in := #Mode_Write, out1 => #statMBMasterBuffer[1].MODE)
   END_RUNG
   RUNG wire#w2
      Move(in := #Addr_TempPV, out1 => #statMBMasterBuffer[1].DATA_ADDR)
      Move(in := 1, out1 => #statMBMasterBuffer[1].DATA_LEN)
   END_RUNG
   RUNG wire#w2
      Move(in := #CMD_Run, out1 => #statMBMasterBuffer[1].DataPTR[1])
      Coil( #"statE5CC[1]".statWriteReq[0] )
   END_RUNG
   RUNG wire#w1
      N_Contact(operand := #statMBMasterBuffer[1].DONE, bit := #statPulse[12])
      R_Coil( #"statE5CC[1]".statWriteReq[0] )
   END_RUNG
   // the same network as SCL:
   #_w1 := #enable AND NOT #"statE5CC[1]".statWriteReq[9] AND #statCMDKeep."E5CC[1]".Upper_Heater_Run;
   IF #_w1 THEN
       #statMBMasterBuffer[1].MB_ADDR := 1;
       #statMBMasterBuffer[1].MODE := #Mode_Write;
       #statMBMasterBuffer[1].DATA_ADDR := #Addr_TempPV;
       #statMBMasterBuffer[1].DATA_LEN := 1;
       #statMBMasterBuffer[1].DataPTR[1] := #CMD_Run;
   END_IF;
   #"statE5CC[1]".statWriteReq[0] := #_w1;
   #_w2 := #enable AND NOT #statMBMasterBuffer[1].DONE AND #statPulse[12];   // falling edge of #statMBMasterBuffer[1].DONE
   #statPulse[12] := #statMBMasterBuffer[1].DONE;
   IF #_w2 THEN #"statE5CC[1]".statWriteReq[0] := FALSE; END_IF;
END_REGION

REGION Network 11: E5CC[1] -Write Heater Stop Command
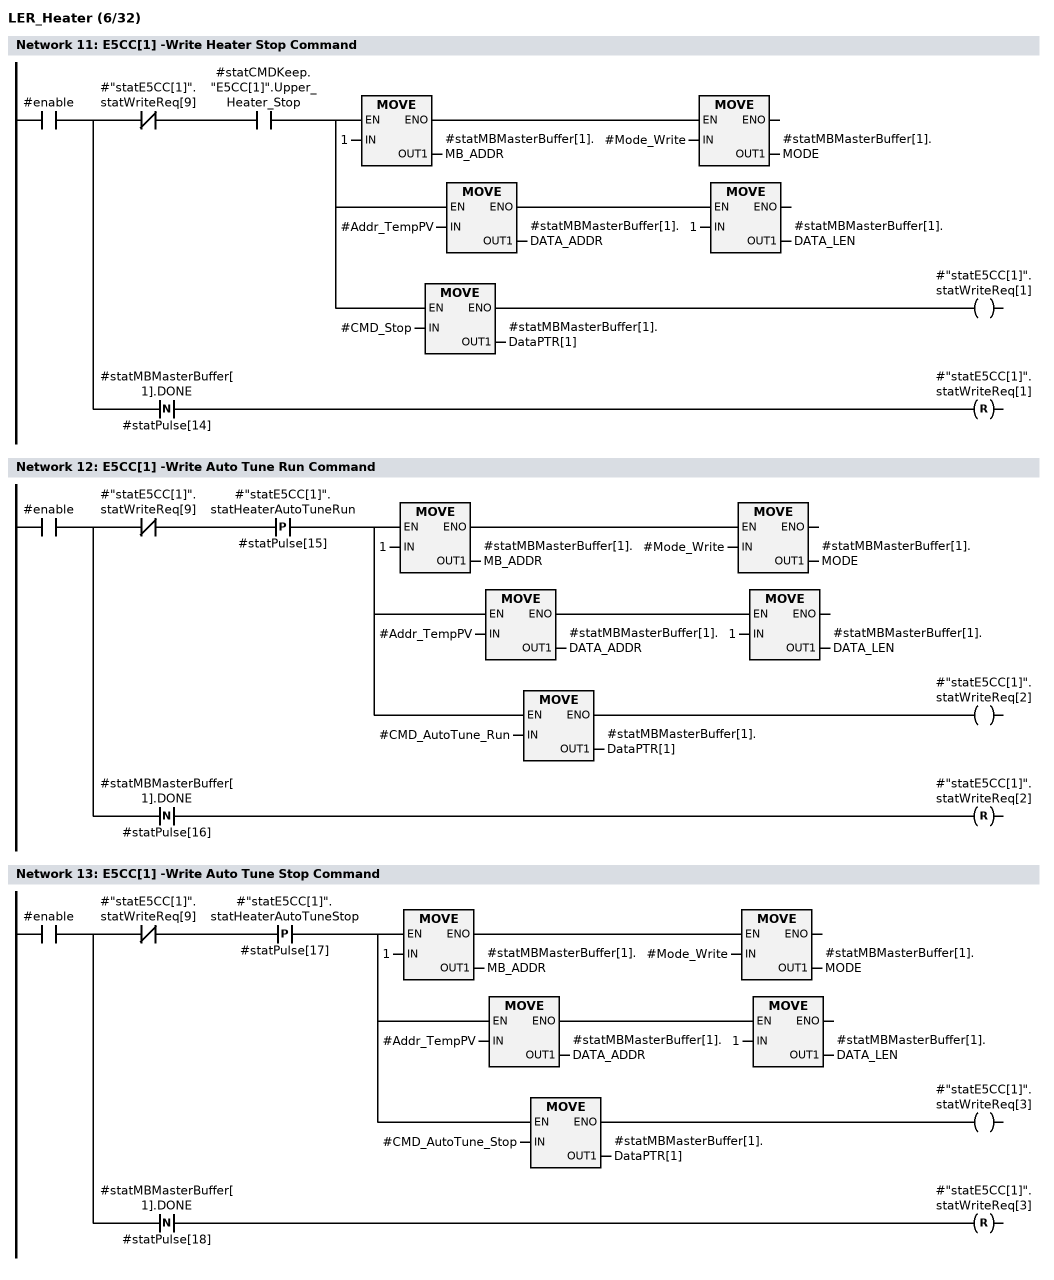
   RUNG wire#powerrail
      Contact( #enable )
      wire#w1
      I_Contact( #"statE5CC[1]".statWriteReq[9] )
      Contact( #statCMDKeep."E5CC[1]".Upper_Heater_Stop )
      wire#w2
      Move(in := 1, out1 => #statMBMasterBuffer[1].MB_ADDR)
      Move(in := #Mode_Write, out1 => #statMBMasterBuffer[1].MODE)
   END_RUNG
   RUNG wire#w2
      Move(in := #Addr_TempPV, out1 => #statMBMasterBuffer[1].DATA_ADDR)
      Move(in := 1, out1 => #statMBMasterBuffer[1].DATA_LEN)
   END_RUNG
   RUNG wire#w2
      Move(in := #CMD_Stop, out1 => #statMBMasterBuffer[1].DataPTR[1])
      Coil( #"statE5CC[1]".statWriteReq[1] )
   END_RUNG
   RUNG wire#w1
      N_Contact(operand := #statMBMasterBuffer[1].DONE, bit := #statPulse[14])
      R_Coil( #"statE5CC[1]".statWriteReq[1] )
   END_RUNG
   // the same network as SCL:
   #_w1 := #enable AND NOT #"statE5CC[1]".statWriteReq[9] AND #statCMDKeep."E5CC[1]".Upper_Heater_Stop;
   IF #_w1 THEN
       #statMBMasterBuffer[1].MB_ADDR := 1;
       #statMBMasterBuffer[1].MODE := #Mode_Write;
       #statMBMasterBuffer[1].DATA_ADDR := #Addr_TempPV;
       #statMBMasterBuffer[1].DATA_LEN := 1;
       #statMBMasterBuffer[1].DataPTR[1] := #CMD_Stop;
   END_IF;
   #"statE5CC[1]".statWriteReq[1] := #_w1;
   #_w2 := #enable AND NOT #statMBMasterBuffer[1].DONE AND #statPulse[14];   // falling edge of #statMBMasterBuffer[1].DONE
   #statPulse[14] := #statMBMasterBuffer[1].DONE;
   IF #_w2 THEN #"statE5CC[1]".statWriteReq[1] := FALSE; END_IF;
END_REGION

REGION Network 12: E5CC[1] -Write Auto Tune Run Command
   RUNG wire#powerrail
      Contact( #enable )
      wire#w1
      I_Contact( #"statE5CC[1]".statWriteReq[9] )
      P_Contact(operand := #"statE5CC[1]".statHeaterAutoTuneRun, bit := #statPulse[15])
      wire#w2
      Move(in := 1, out1 => #statMBMasterBuffer[1].MB_ADDR)
      Move(in := #Mode_Write, out1 => #statMBMasterBuffer[1].MODE)
   END_RUNG
   RUNG wire#w2
      Move(in := #Addr_TempPV, out1 => #statMBMasterBuffer[1].DATA_ADDR)
      Move(in := 1, out1 => #statMBMasterBuffer[1].DATA_LEN)
   END_RUNG
   RUNG wire#w2
      Move(in := #CMD_AutoTune_Run, out1 => #statMBMasterBuffer[1].DataPTR[1])
      Coil( #"statE5CC[1]".statWriteReq[2] )
   END_RUNG
   RUNG wire#w1
      N_Contact(operand := #statMBMasterBuffer[1].DONE, bit := #statPulse[16])
      R_Coil( #"statE5CC[1]".statWriteReq[2] )
   END_RUNG
   // the same network as SCL:
   #_w1 := #enable AND NOT #"statE5CC[1]".statWriteReq[9] AND #"statE5CC[1]".statHeaterAutoTuneRun AND NOT #statPulse[15];   // rising edge of #"statE5CC[1]".statHeaterAutoTuneRun
   #statPulse[15] := #"statE5CC[1]".statHeaterAutoTuneRun;
   IF #_w1 THEN
       #statMBMasterBuffer[1].MB_ADDR := 1;
       #statMBMasterBuffer[1].MODE := #Mode_Write;
       #statMBMasterBuffer[1].DATA_ADDR := #Addr_TempPV;
       #statMBMasterBuffer[1].DATA_LEN := 1;
       #statMBMasterBuffer[1].DataPTR[1] := #CMD_AutoTune_Run;
   END_IF;
   #"statE5CC[1]".statWriteReq[2] := #_w1;
   #_w2 := #enable AND NOT #statMBMasterBuffer[1].DONE AND #statPulse[16];   // falling edge of #statMBMasterBuffer[1].DONE
   #statPulse[16] := #statMBMasterBuffer[1].DONE;
   IF #_w2 THEN #"statE5CC[1]".statWriteReq[2] := FALSE; END_IF;
END_REGION

REGION Network 13: E5CC[1] -Write Auto Tune Stop Command
   RUNG wire#powerrail
      Contact( #enable )
      wire#w1
      I_Contact( #"statE5CC[1]".statWriteReq[9] )
      P_Contact(operand := #"statE5CC[1]".statHeaterAutoTuneStop, bit := #statPulse[17])
      wire#w2
      Move(in := 1, out1 => #statMBMasterBuffer[1].MB_ADDR)
      Move(in := #Mode_Write, out1 => #statMBMasterBuffer[1].MODE)
   END_RUNG
   RUNG wire#w2
      Move(in := #Addr_TempPV, out1 => #statMBMasterBuffer[1].DATA_ADDR)
      Move(in := 1, out1 => #statMBMasterBuffer[1].DATA_LEN)
   END_RUNG
   RUNG wire#w2
      Move(in := #CMD_AutoTune_Stop, out1 => #statMBMasterBuffer[1].DataPTR[1])
      Coil( #"statE5CC[1]".statWriteReq[3] )
   END_RUNG
   RUNG wire#w1
      N_Contact(operand := #statMBMasterBuffer[1].DONE, bit := #statPulse[18])
      R_Coil( #"statE5CC[1]".statWriteReq[3] )
   END_RUNG
   // the same network as SCL:
   #_w1 := #enable AND NOT #"statE5CC[1]".statWriteReq[9] AND #"statE5CC[1]".statHeaterAutoTuneStop AND NOT #statPulse[17];   // rising edge of #"statE5CC[1]".statHeaterAutoTuneStop
   #statPulse[17] := #"statE5CC[1]".statHeaterAutoTuneStop;
   IF #_w1 THEN
       #statMBMasterBuffer[1].MB_ADDR := 1;
       #statMBMasterBuffer[1].MODE := #Mode_Write;
       #statMBMasterBuffer[1].DATA_ADDR := #Addr_TempPV;
       #statMBMasterBuffer[1].DATA_LEN := 1;
       #statMBMasterBuffer[1].DataPTR[1] := #CMD_AutoTune_Stop;
   END_IF;
   #"statE5CC[1]".statWriteReq[3] := #_w1;
   #_w2 := #enable AND NOT #statMBMasterBuffer[1].DONE AND #statPulse[18];   // falling edge of #statMBMasterBuffer[1].DONE
   #statPulse[18] := #statMBMasterBuffer[1].DONE;
   IF #_w2 THEN #"statE5CC[1]".statWriteReq[3] := FALSE; END_IF;
END_REGION

REGION Network 14: E5CC[1] -Write TempSP + AlarmValue1 ~ AlarmValue2_LowerLimit Command
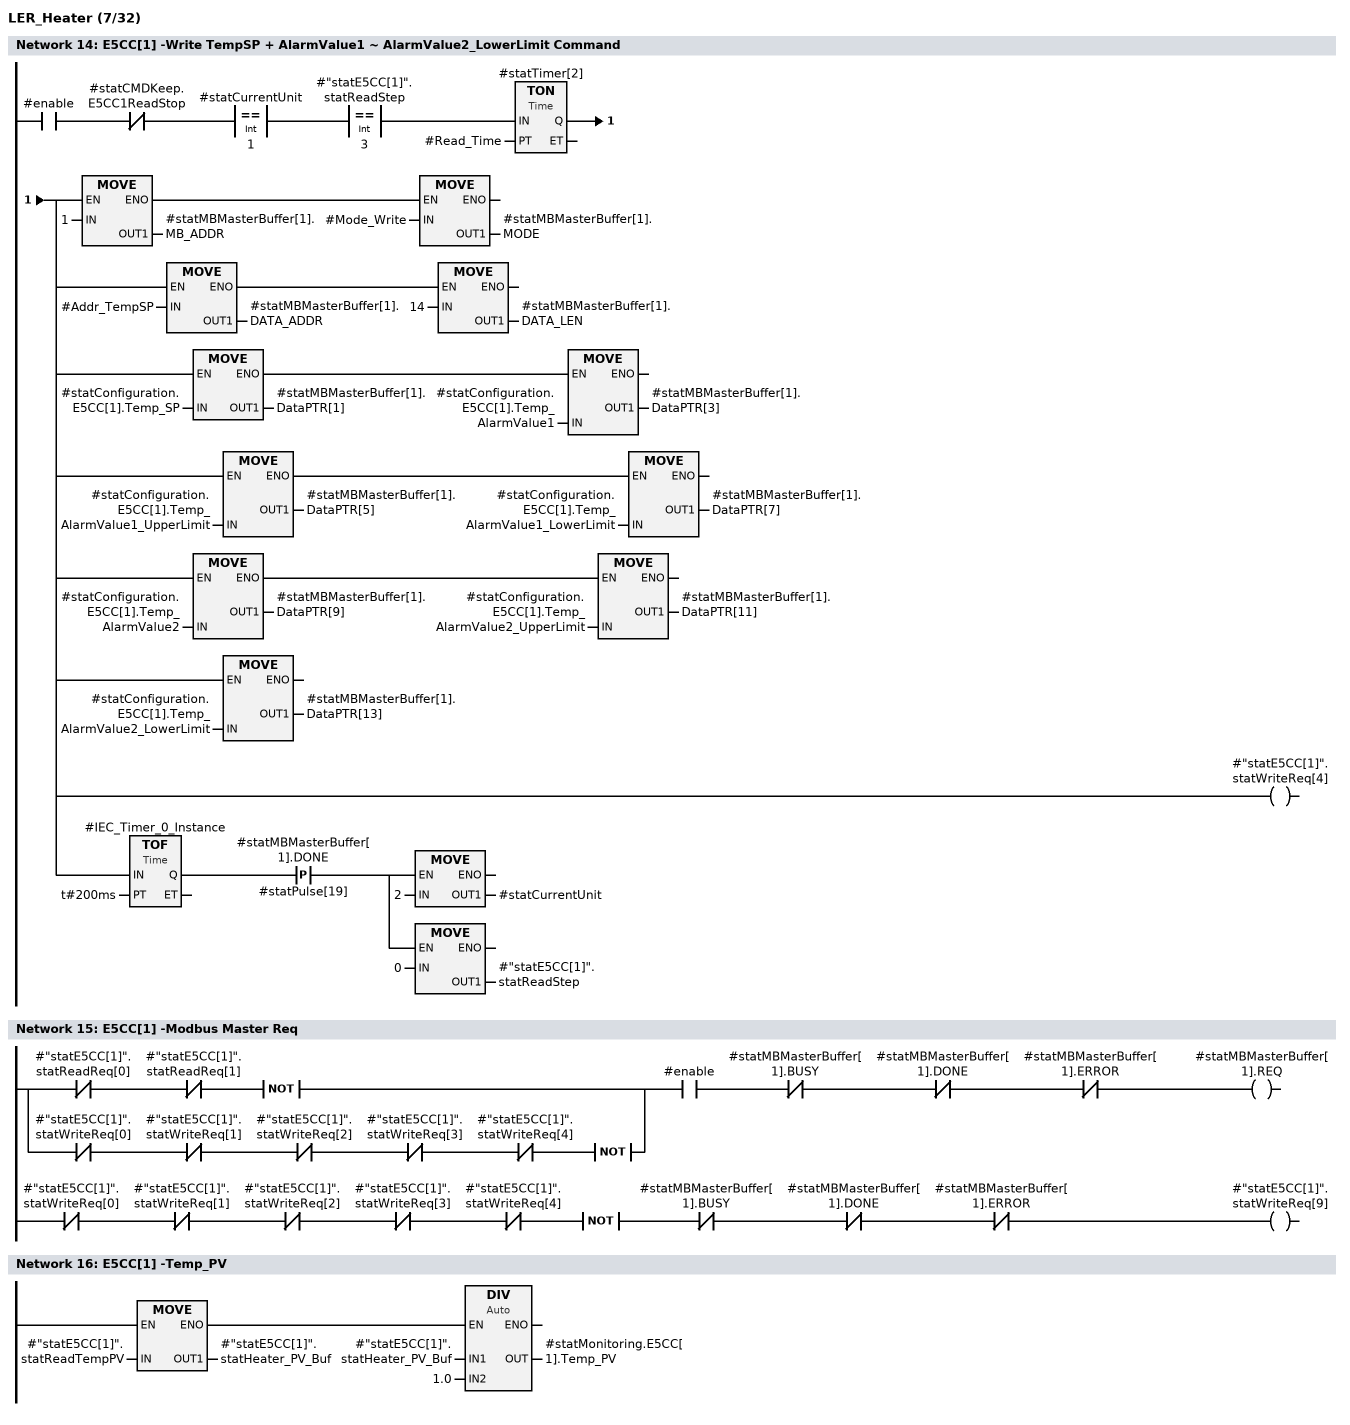
   RUNG wire#powerrail
      Contact( #enable )
      I_Contact( #statCMDKeep.E5CC1ReadStop )
      { S7_Templates := "SrcType := Int" } EQ_Contact(in1 := #statCurrentUnit, in2 := 1)
      { S7_Templates := "SrcType := Int" } EQ_Contact(in1 := #"statE5CC[1]".statReadStep, in2 := 3)
      { S7_Templates := "time_type := Time" } #statTimer[2].TON(pt := #Read_Time, et =>)
      wire#w1
      Move(in := 1, out1 => #statMBMasterBuffer[1].MB_ADDR)
      Move(in := #Mode_Write, out1 => #statMBMasterBuffer[1].MODE)
   END_RUNG
   RUNG wire#w1
      Move(in := #Addr_TempSP, out1 => #statMBMasterBuffer[1].DATA_ADDR)
      Move(in := 14, out1 => #statMBMasterBuffer[1].DATA_LEN)
   END_RUNG
   RUNG wire#w1
      Move(in := #statConfiguration.E5CC[1].Temp_SP, out1 => #statMBMasterBuffer[1].DataPTR[1])
      Move(in := #statConfiguration.E5CC[1].Temp_AlarmValue1, out1 => #statMBMasterBuffer[1].DataPTR[3])
   END_RUNG
   RUNG wire#w1
      Move(in := #statConfiguration.E5CC[1].Temp_AlarmValue1_UpperLimit, out1 => #statMBMasterBuffer[1].DataPTR[5])
      Move(in := #statConfiguration.E5CC[1].Temp_AlarmValue1_LowerLimit, out1 => #statMBMasterBuffer[1].DataPTR[7])
   END_RUNG
   RUNG wire#w1
      Move(in := #statConfiguration.E5CC[1].Temp_AlarmValue2, out1 => #statMBMasterBuffer[1].DataPTR[9])
      Move(in := #statConfiguration.E5CC[1].Temp_AlarmValue2_UpperLimit, out1 => #statMBMasterBuffer[1].DataPTR[11])
   END_RUNG
   RUNG wire#w1
      Move(in := #statConfiguration.E5CC[1].Temp_AlarmValue2_LowerLimit, out1 => #statMBMasterBuffer[1].DataPTR[13])
   END_RUNG
   RUNG wire#w1
      Coil( #"statE5CC[1]".statWriteReq[4] )
   END_RUNG
   RUNG wire#w1
      { S7_Templates := "time_type := Time" } #IEC_Timer_0_Instance.TOF(pt := t#200ms, et =>)
      P_Contact(operand := #statMBMasterBuffer[1].DONE, bit := #statPulse[19])
      wire#w2
      Move(in := 2, out1 => #statCurrentUnit)
   END_RUNG
   RUNG wire#w2
      Move(in := 0, out1 => #"statE5CC[1]".statReadStep)
   END_RUNG
   // the same network as SCL:
   #statTimer[2].TON(IN := #enable AND NOT #statCMDKeep.E5CC1ReadStop AND (#statCurrentUnit = 1) AND (#"statE5CC[1]".statReadStep = 3),
                     PT := #Read_Time);
   IF #statTimer[2].Q THEN
       #statMBMasterBuffer[1].MB_ADDR := 1;
       #statMBMasterBuffer[1].MODE := #Mode_Write;
       #statMBMasterBuffer[1].DATA_ADDR := #Addr_TempSP;
       #statMBMasterBuffer[1].DATA_LEN := 14;
       #statMBMasterBuffer[1].DataPTR[1] := #statConfiguration.E5CC[1].Temp_SP;
       #statMBMasterBuffer[1].DataPTR[3] := #statConfiguration.E5CC[1].Temp_AlarmValue1;
       #statMBMasterBuffer[1].DataPTR[5] := #statConfiguration.E5CC[1].Temp_AlarmValue1_UpperLimit;
       #statMBMasterBuffer[1].DataPTR[7] := #statConfiguration.E5CC[1].Temp_AlarmValue1_LowerLimit;
       #statMBMasterBuffer[1].DataPTR[9] := #statConfiguration.E5CC[1].Temp_AlarmValue2;
       #statMBMasterBuffer[1].DataPTR[11] := #statConfiguration.E5CC[1].Temp_AlarmValue2_UpperLimit;
       #statMBMasterBuffer[1].DataPTR[13] := #statConfiguration.E5CC[1].Temp_AlarmValue2_LowerLimit;
   END_IF;
   #"statE5CC[1]".statWriteReq[4] := #statTimer[2].Q;
   #IEC_Timer_0_Instance(IN := #statTimer[2].Q, PT := t#200ms);   // TOF
   #_w1 := #IEC_Timer_0_Instance.Q AND #statMBMasterBuffer[1].DONE AND NOT #statPulse[19];   // rising edge of #statMBMasterBuffer[1].DONE
   #statPulse[19] := #statMBMasterBuffer[1].DONE;
   IF #_w1 THEN
       #statCurrentUnit := 2;
       #"statE5CC[1]".statReadStep := 0;
   END_IF;
END_REGION

REGION Network 15: E5CC[1] -Modbus Master Req
   RUNG wire#powerrail
      I_Contact( #"statE5CC[1]".statReadReq[0] )
      I_Contact( #"statE5CC[1]".statReadReq[1] )
      Not()
      wire#w1
      Contact( #enable )
      I_Contact( #statMBMasterBuffer[1].BUSY )
      I_Contact( #statMBMasterBuffer[1].DONE )
      I_Contact( #statMBMasterBuffer[1].ERROR )
      Coil( #statMBMasterBuffer[1].REQ )
   END_RUNG
   RUNG wire#powerrail
      I_Contact( #"statE5CC[1]".statWriteReq[0] )
      I_Contact( #"statE5CC[1]".statWriteReq[1] )
      I_Contact( #"statE5CC[1]".statWriteReq[2] )
      I_Contact( #"statE5CC[1]".statWriteReq[3] )
      I_Contact( #"statE5CC[1]".statWriteReq[4] )
      Not()
   END_RUNG wire#w1
   RUNG wire#powerrail
      I_Contact( #"statE5CC[1]".statWriteReq[0] )
      I_Contact( #"statE5CC[1]".statWriteReq[1] )
      I_Contact( #"statE5CC[1]".statWriteReq[2] )
      I_Contact( #"statE5CC[1]".statWriteReq[3] )
      I_Contact( #"statE5CC[1]".statWriteReq[4] )
      Not()
      I_Contact( #statMBMasterBuffer[1].BUSY )
      I_Contact( #statMBMasterBuffer[1].DONE )
      I_Contact( #statMBMasterBuffer[1].ERROR )
      Coil( #"statE5CC[1]".statWriteReq[9] )
   END_RUNG
   // the same network as SCL:
   #statMBMasterBuffer[1].REQ := (NOT (NOT #"statE5CC[1]".statReadReq[0] AND NOT #"statE5CC[1]".statReadReq[1]) OR NOT (NOT #"statE5CC[1]".statWriteReq[0] AND NOT #"statE5CC[1]".statWriteReq[1] AND NOT #"statE5CC[1]".statWriteReq[2] AND NOT #"statE5CC[1]".statWriteReq[3] AND NOT #"statE5CC[1]".statWriteReq[4])) AND #enable AND NOT #statMBMasterBuffer[1].BUSY AND NOT #statMBMasterBuffer[1].DONE AND NOT #statMBMasterBuffer[1].ERROR;
   #"statE5CC[1]".statWriteReq[9] := NOT (NOT #"statE5CC[1]".statWriteReq[0] AND NOT #"statE5CC[1]".statWriteReq[1] AND NOT #"statE5CC[1]".statWriteReq[2] AND NOT #"statE5CC[1]".statWriteReq[3] AND NOT #"statE5CC[1]".statWriteReq[4]) AND NOT #statMBMasterBuffer[1].BUSY AND NOT #statMBMasterBuffer[1].DONE AND NOT #statMBMasterBuffer[1].ERROR;
END_REGION

REGION Network 16: E5CC[1] -Temp_PV
   RUNG wire#powerrail
      Move(in := #"statE5CC[1]".statReadTempPV, out1 => #"statE5CC[1]".statHeater_PV_Buf)
      Div(in1 := #"statE5CC[1]".statHeater_PV_Buf, in2 := 1.0, out => #statMonitoring.E5CC[1].Temp_PV)
   END_RUNG
   // the same network as SCL:
   #"statE5CC[1]".statHeater_PV_Buf := #"statE5CC[1]".statReadTempPV;
   #statMonitoring.E5CC[1].Temp_PV := #"statE5CC[1]".statHeater_PV_Buf / 1.0;
END_REGION

REGION Network 17: E5CC[1] -Temp_PV Complete Check
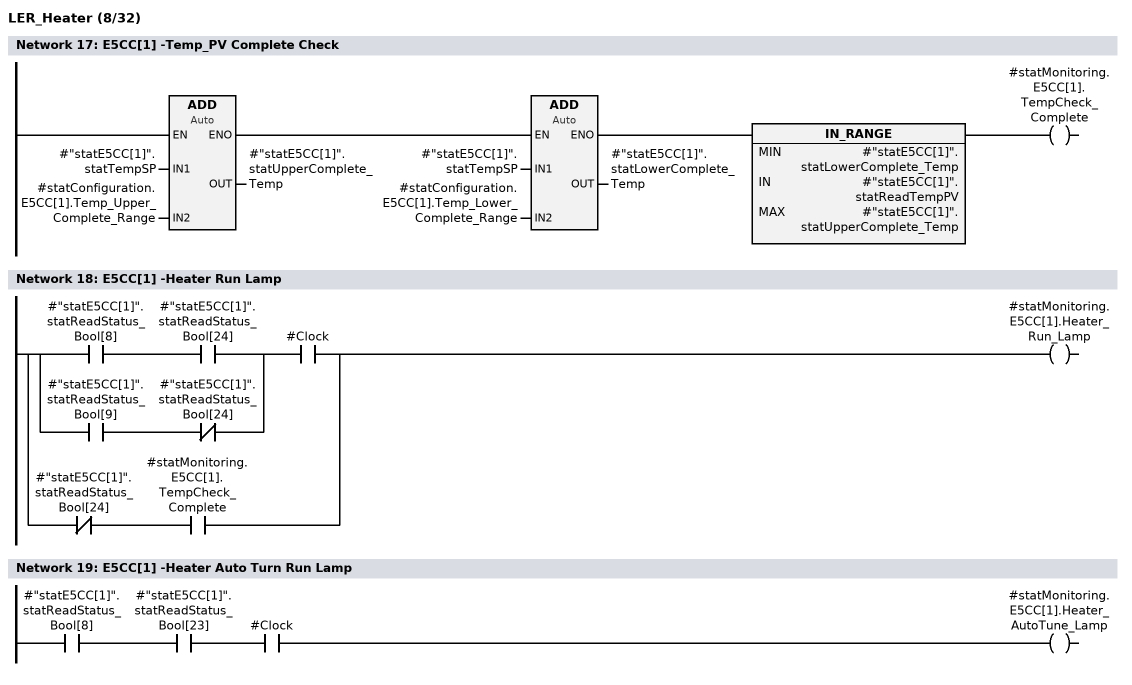
   RUNG wire#powerrail
      Add(in1 := #"statE5CC[1]".statTempSP, in2 := #statConfiguration.E5CC[1].Temp_Upper_Complete_Range, out => #"statE5CC[1]".statUpperComplete_Temp)
      Add(in1 := #"statE5CC[1]".statTempSP, in2 := #statConfiguration.E5CC[1].Temp_Lower_Complete_Range, out => #"statE5CC[1]".statLowerComplete_Temp)
      { S7_Templates := "SrcType := Real" } InRange(min := #"statE5CC[1]".statLowerComplete_Temp, in := #"statE5CC[1]".statReadTempPV, max := #"statE5CC[1]".statUpperComplete_Temp)
      Coil( #statMonitoring.E5CC[1].TempCheck_Complete )
   END_RUNG
   // the same network as SCL:
   #"statE5CC[1]".statUpperComplete_Temp := #"statE5CC[1]".statTempSP + #statConfiguration.E5CC[1].Temp_Upper_Complete_Range;
   #"statE5CC[1]".statLowerComplete_Temp := #"statE5CC[1]".statTempSP + #statConfiguration.E5CC[1].Temp_Lower_Complete_Range;
   #statMonitoring.E5CC[1].TempCheck_Complete := (#"statE5CC[1]".statLowerComplete_Temp <= #"statE5CC[1]".statReadTempPV) AND (#"statE5CC[1]".statReadTempPV <= #"statE5CC[1]".statUpperComplete_Temp);
END_REGION

REGION Network 18: E5CC[1] -Heater Run Lamp
   RUNG wire#powerrail
      Contact( #"statE5CC[1]".statReadStatus_Bool[8] )
      Contact( #"statE5CC[1]".statReadStatus_Bool[24] )
      wire#w1
      Contact( #Clock )
      wire#w2
      Coil( #statMonitoring.E5CC[1].Heater_Run_Lamp )
   END_RUNG
   RUNG wire#powerrail
      Contact( #"statE5CC[1]".statReadStatus_Bool[9] )
      I_Contact( #"statE5CC[1]".statReadStatus_Bool[24] )
   END_RUNG wire#w1
   RUNG wire#powerrail
      I_Contact( #"statE5CC[1]".statReadStatus_Bool[24] )
      Contact( #statMonitoring.E5CC[1].TempCheck_Complete )
   END_RUNG wire#w2
   // the same network as SCL:
   #statMonitoring.E5CC[1].Heater_Run_Lamp := (((#"statE5CC[1]".statReadStatus_Bool[8] AND #"statE5CC[1]".statReadStatus_Bool[24]) OR (#"statE5CC[1]".statReadStatus_Bool[9] AND NOT #"statE5CC[1]".statReadStatus_Bool[24])) AND #Clock) OR (NOT #"statE5CC[1]".statReadStatus_Bool[24] AND #statMonitoring.E5CC[1].TempCheck_Complete);
END_REGION

REGION Network 19: E5CC[1] -Heater Auto Turn Run Lamp
   RUNG wire#powerrail
      Contact( #"statE5CC[1]".statReadStatus_Bool[8] )
      Contact( #"statE5CC[1]".statReadStatus_Bool[23] )
      Contact( #Clock )
      Coil( #statMonitoring.E5CC[1].Heater_AutoTune_Lamp )
   END_RUNG
   // the same network as SCL:
   #statMonitoring.E5CC[1].Heater_AutoTune_Lamp := #"statE5CC[1]".statReadStatus_Bool[8] AND #"statE5CC[1]".statReadStatus_Bool[23] AND #Clock;
END_REGION

REGION Network 20 (SCL): E5CC[1] -Error Check
   REGION  E5CC Error Status
       // Dword to Bool
       SCATTER(IN := #"statE5CC[1]".statReadStatus,
               OUT => #"statE5CC[1]".statReadStatus_Bool);
   END_REGION


   REGION Error Code Search
       IF #"statE5CC[1]".statReadStatus <> 0 THEN
           CASE #"statE5CC[1]".statReadStatus OF
               #ERR_HEATER_CURRENT_VALUE_EXCEEDED_CT1:
                   #statMonitoring.E5CC[1].Status := #ERR_HEATER_CURRENT_VALUE_EXCEEDED_CT1;
               #ERR_HEATER_CURRENT_VALUE_HOLD_CT1:
                   #statMonitoring.E5CC[1].Status := #ERR_HEATER_CURRENT_VALUE_HOLD_CT1;
               #ERR_AD_CONVERTER_ABNORMALITY:
                   #statMonitoring.E5CC[1].Status := #ERR_AD_CONVERTER_ABNORMALITY;
               #ERR_HS_SSR_FAULT_ALERT_CT1:
                   #statMonitoring.E5CC[1].Status := #ERR_HS_SSR_FAULT_ALERT_CT1;
               #ERR_RSP_INPUT_ABNORMALITIES:
                   #statMonitoring.E5CC[1].Status := #ERR_RSP_INPUT_ABNORMALITIES;
               #ERR_MORE_THAN_INPUT:
                   #statMonitoring.E5CC[1].Status := #ERR_MORE_THAN_INPUT;
               #ERR_POTENTIOMETER_INPUT_ABNORMAL:
                   #statMonitoring.E5CC[1].Status := #ERR_POTENTIOMETER_INPUT_ABNORMAL;
               #ERR_CONTROL_OUTPUT_HEATED_OPEN_OUTPUT:
                   #statMonitoring.E5CC[1].Status := #ERR_CONTROL_OUTPUT_HEATED_OPEN_OUTPUT;
               #ERR_CONTROL_OUTPUT_COOL_CLOSE_OUTPUT:
                   #statMonitoring.E5CC[1].Status := #ERR_CONTROL_OUTPUT_COOL_CLOSE_OUTPUT;
               #ERR_HEATER_OPEN_CIRCUIT_HB_ALARM_CT1:
                   #statMonitoring.E5CC[1].Status := #ERR_HEATER_OPEN_CIRCUIT_HB_ALARM_CT1;
               #ERR_HEATER_OPEN_CIRCUIT_HB_ALARM_CT2:
                   #statMonitoring.E5CC[1].Status := #ERR_HEATER_OPEN_CIRCUIT_HB_ALARM_CT2;
               #ERR_ALERT_1:
                   #statMonitoring.E5CC[1].Status := #ERR_ALERT_1;
               #ERR_ALERT_2:
                   #statMonitoring.E5CC[1].Status := #ERR_ALERT_2;
               #ERR_ALERT_3:
                   #statMonitoring.E5CC[1].Status := #ERR_ALERT_3;
               #ERR_PROGRAM_END_OUTPUT:
                   #statMonitoring.E5CC[1].Status := #ERR_PROGRAM_END_OUTPUT;
               #ERR_EVENT_INPUT_1:
                   #statMonitoring.E5CC[1].Status := #ERR_EVENT_INPUT_1;
               #ERR_EVENT_INPUT_2:
                   #statMonitoring.E5CC[1].Status := #ERR_EVENT_INPUT_2;
               #ERR_EVENT_INPUT_3:
                   #statMonitoring.E5CC[1].Status := #ERR_EVENT_INPUT_3;
               #ERR_EVENT_INPUT_4:
                   #statMonitoring.E5CC[1].Status := #ERR_EVENT_INPUT_4;
               #ERR_WRITE_MODE:
                   #statMonitoring.E5CC[1].Status := #ERR_WRITE_MODE;
               #ERR_NON_VOLATILE_MEMORY:
                   #statMonitoring.E5CC[1].Status := #ERR_NON_VOLATILE_MEMORY;
               #ERR_SETTING_AREA:
                   #statMonitoring.E5CC[1].Status := #ERR_SETTING_AREA;
               #ERR_AT_RUN_STOP:
                   #statMonitoring.E5CC[1].Status := #ERR_AT_RUN_STOP;
               #ERR_RUN_STOP:
                   #statMonitoring.E5CC[1].Status := #ERR_RUN_STOP;
               #ERR_COMMUNICATION_WRITE:
                   #statMonitoring.E5CC[1].Status := #ERR_COMMUNICATION_WRITE;
               #ERR_AUTO_MANUAL:
                   #statMonitoring.E5CC[1].Status := #ERR_AUTO_MANUAL;
               #ERR_PROGRAM_START:
                   #statMonitoring.E5CC[1].Status := #ERR_PROGRAM_START;
               #ERR_HEATER_CURRENT_VALUE_EXCEEDED_CT2:
                   #statMonitoring.E5CC[1].Status := #ERR_HEATER_CURRENT_VALUE_EXCEEDED_CT2;
               #ERR_HEATER_CURRENT_VALUE_HOLD_CT2:
                   #statMonitoring.E5CC[1].Status := #ERR_HEATER_CURRENT_VALUE_HOLD_CT2;
               #ERR_HS_SSR_FAILURE_ALARM_CT2:
                   #statMonitoring.E5CC[1].Status := #ERR_HS_SSR_FAILURE_ALARM_CT2;
           END_CASE;
       ELSIF #"statE5CC[1]".statReadStatus = 0 THEN
           #statMonitoring.E5CC[1].Status := 0;
       END_IF;
   END_REGION

   #statMonitoring.E5CC[1].Error := #"statE5CC[1]".statReadStatus <> 0;
END_REGION

REGION Network 21 (SCL): E5CC[1] -##### Outputs mapping #####
   // Output Mapping
   #statMonitoring.E5CC[1].Temp_SP := #"statE5CC[1]".statTempSP;
   #statMonitoring.E5CC[1].Temp_AlarmValue1 := #"statE5CC[1]".statAlarmValue1;
   #statMonitoring.E5CC[1].Temp_AlarmValue1_UpperLimit := #"statE5CC[1]".statAlarmValue1_UpperLimit;
   #statMonitoring.E5CC[1].Temp_AlarmValue1_LowerLimit := #"statE5CC[1]".statAlarmValue1_LowerLimit;
   #statMonitoring.E5CC[1].Temp_AlarmValue2 := #"statE5CC[1]".statAlarmValue2;
   #statMonitoring.E5CC[1].Temp_AlarmValue2_UpperLimit := #"statE5CC[1]".statAlarmValue2_UpperLimit;
   #statMonitoring.E5CC[1].Temp_AlarmValue2_LowerLimit := #"statE5CC[1]".statAlarmValue2_LowerLimit;
   #statMonitoring.E5CC[1].E5CC_Status := #"statE5CC[1]".statReadStatus;
   #statMonitoring.E5CC[1].E5CC_Status_Bool := #"statE5CC[1]".statReadStatus_Bool;
END_REGION

REGION Network 22: E5CC[2] - ###### Input Mapping ######
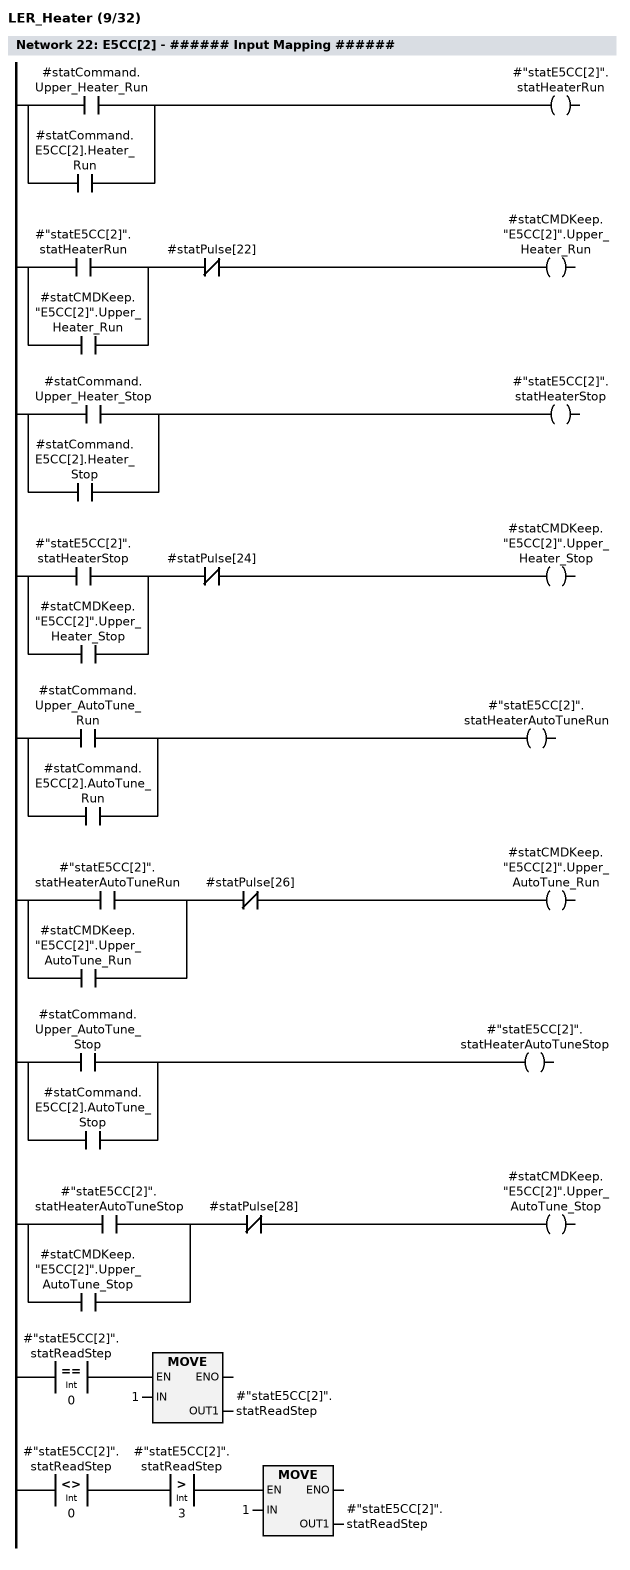
   RUNG wire#powerrail
      Contact( #statCommand.Upper_Heater_Run )
      wire#w1
      Coil( #"statE5CC[2]".statHeaterRun )
   END_RUNG
   RUNG wire#powerrail
      Contact( #statCommand.E5CC[2].Heater_Run )
   END_RUNG wire#w1
   RUNG wire#powerrail
      Contact( #"statE5CC[2]".statHeaterRun )
      wire#w2
      I_Contact( #statPulse[22] )
      Coil( #statCMDKeep."E5CC[2]".Upper_Heater_Run )
   END_RUNG
   RUNG wire#powerrail
      Contact( #statCMDKeep."E5CC[2]".Upper_Heater_Run )
   END_RUNG wire#w2
   RUNG wire#powerrail
      Contact( #statCommand.Upper_Heater_Stop )
      wire#w3
      Coil( #"statE5CC[2]".statHeaterStop )
   END_RUNG
   RUNG wire#powerrail
      Contact( #statCommand.E5CC[2].Heater_Stop )
   END_RUNG wire#w3
   RUNG wire#powerrail
      Contact( #"statE5CC[2]".statHeaterStop )
      wire#w4
      I_Contact( #statPulse[24] )
      Coil( #statCMDKeep."E5CC[2]".Upper_Heater_Stop )
   END_RUNG
   RUNG wire#powerrail
      Contact( #statCMDKeep."E5CC[2]".Upper_Heater_Stop )
   END_RUNG wire#w4
   RUNG wire#powerrail
      Contact( #statCommand.Upper_AutoTune_Run )
      wire#w5
      Coil( #"statE5CC[2]".statHeaterAutoTuneRun )
   END_RUNG
   RUNG wire#powerrail
      Contact( #statCommand.E5CC[2].AutoTune_Run )
   END_RUNG wire#w5
   RUNG wire#powerrail
      Contact( #"statE5CC[2]".statHeaterAutoTuneRun )
      wire#w6
      I_Contact( #statPulse[26] )
      Coil( #statCMDKeep."E5CC[2]".Upper_AutoTune_Run )
   END_RUNG
   RUNG wire#powerrail
      Contact( #statCMDKeep."E5CC[2]".Upper_AutoTune_Run )
   END_RUNG wire#w6
   RUNG wire#powerrail
      Contact( #statCommand.Upper_AutoTune_Stop )
      wire#w7
      Coil( #"statE5CC[2]".statHeaterAutoTuneStop )
   END_RUNG
   RUNG wire#powerrail
      Contact( #statCommand.E5CC[2].AutoTune_Stop )
   END_RUNG wire#w7
   RUNG wire#powerrail
      Contact( #"statE5CC[2]".statHeaterAutoTuneStop )
      wire#w8
      I_Contact( #statPulse[28] )
      Coil( #statCMDKeep."E5CC[2]".Upper_AutoTune_Stop )
   END_RUNG
   RUNG wire#powerrail
      Contact( #statCMDKeep."E5CC[2]".Upper_AutoTune_Stop )
   END_RUNG wire#w8
   RUNG wire#powerrail
      { S7_Templates := "SrcType := Int" } EQ_Contact(in1 := #"statE5CC[2]".statReadStep, in2 := 0)
      Move(in := 1, out1 => #"statE5CC[2]".statReadStep)
   END_RUNG
   RUNG wire#powerrail
      { S7_Templates := "SrcType := Int" } NE_Contact(in1 := #"statE5CC[2]".statReadStep, in2 := 0)
      { S7_Templates := "SrcType := Int" } GT_Contact(in1 := #"statE5CC[2]".statReadStep, in2 := 3)
      Move(in := 1, out1 => #"statE5CC[2]".statReadStep)
   END_RUNG
   // the same network as SCL:
   #"statE5CC[2]".statHeaterRun := #statCommand.Upper_Heater_Run OR #statCommand.E5CC[2].Heater_Run;
   #statCMDKeep."E5CC[2]".Upper_Heater_Run := (#"statE5CC[2]".statHeaterRun OR #statCMDKeep."E5CC[2]".Upper_Heater_Run) AND NOT #statPulse[22];
   #"statE5CC[2]".statHeaterStop := #statCommand.Upper_Heater_Stop OR #statCommand.E5CC[2].Heater_Stop;
   #statCMDKeep."E5CC[2]".Upper_Heater_Stop := (#"statE5CC[2]".statHeaterStop OR #statCMDKeep."E5CC[2]".Upper_Heater_Stop) AND NOT #statPulse[24];
   #"statE5CC[2]".statHeaterAutoTuneRun := #statCommand.Upper_AutoTune_Run OR #statCommand.E5CC[2].AutoTune_Run;
   #statCMDKeep."E5CC[2]".Upper_AutoTune_Run := (#"statE5CC[2]".statHeaterAutoTuneRun OR #statCMDKeep."E5CC[2]".Upper_AutoTune_Run) AND NOT #statPulse[26];
   #"statE5CC[2]".statHeaterAutoTuneStop := #statCommand.Upper_AutoTune_Stop OR #statCommand.E5CC[2].AutoTune_Stop;
   #statCMDKeep."E5CC[2]".Upper_AutoTune_Stop := (#"statE5CC[2]".statHeaterAutoTuneStop OR #statCMDKeep."E5CC[2]".Upper_AutoTune_Stop) AND NOT #statPulse[28];
   IF #"statE5CC[2]".statReadStep = 0 THEN #"statE5CC[2]".statReadStep := 1; END_IF;
   IF (#"statE5CC[2]".statReadStep <> 0) AND (#"statE5CC[2]".statReadStep > 3) THEN
       #"statE5CC[2]".statReadStep := 1;
   END_IF;
END_REGION

REGION Network 23: E5CC[2] -Read Temp PV + Status Command
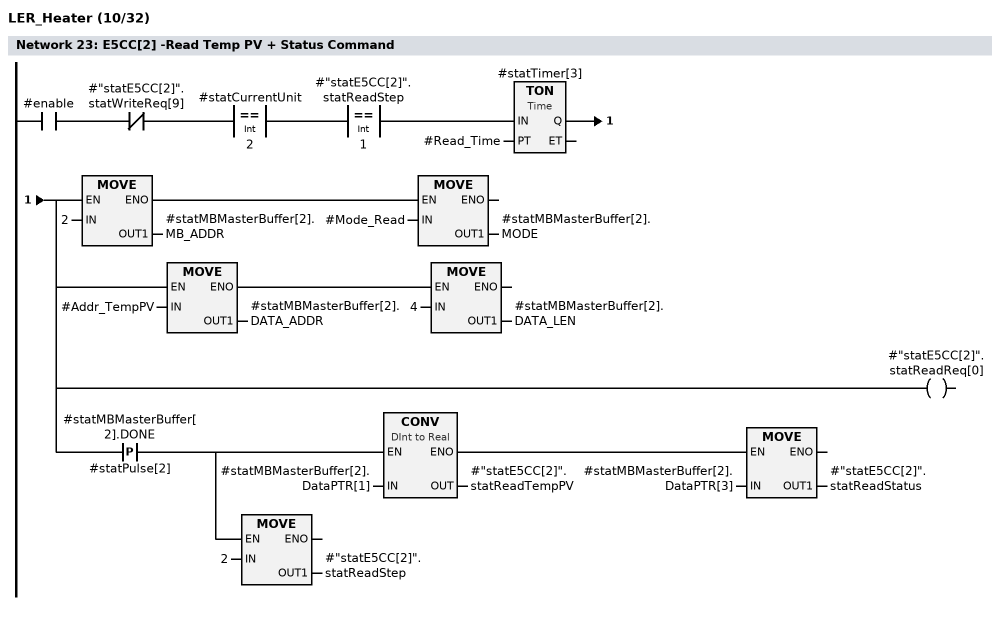
   RUNG wire#powerrail
      Contact( #enable )
      I_Contact( #"statE5CC[2]".statWriteReq[9] )
      { S7_Templates := "SrcType := Int" } EQ_Contact(in1 := #statCurrentUnit, in2 := 2)
      { S7_Templates := "SrcType := Int" } EQ_Contact(in1 := #"statE5CC[2]".statReadStep, in2 := 1)
      { S7_Templates := "time_type := Time" } #statTimer[3].TON(pt := #Read_Time, et =>)
      wire#w1
      Move(in := 2, out1 => #statMBMasterBuffer[2].MB_ADDR)
      Move(in := #Mode_Read, out1 => #statMBMasterBuffer[2].MODE)
   END_RUNG
   RUNG wire#w1
      Move(in := #Addr_TempPV, out1 => #statMBMasterBuffer[2].DATA_ADDR)
      Move(in := 4, out1 => #statMBMasterBuffer[2].DATA_LEN)
   END_RUNG
   RUNG wire#w1
      Coil( #"statE5CC[2]".statReadReq[0] )
   END_RUNG
   RUNG wire#w1
      P_Contact(operand := #statMBMasterBuffer[2].DONE, bit := #statPulse[2])
      wire#w2
      { S7_Templates := "[SrcType := DInt, DestType := Real]" } Convert(in := #statMBMasterBuffer[2].DataPTR[1], out => #"statE5CC[2]".statReadTempPV)
      Move(in := #statMBMasterBuffer[2].DataPTR[3], out1 => #"statE5CC[2]".statReadStatus)
   END_RUNG
   RUNG wire#w2
      Move(in := 2, out1 => #"statE5CC[2]".statReadStep)
   END_RUNG
   // the same network as SCL:
   #statTimer[3].TON(IN := #enable AND NOT #"statE5CC[2]".statWriteReq[9] AND (#statCurrentUnit = 2) AND (#"statE5CC[2]".statReadStep = 1),
                     PT := #Read_Time);
   IF #statTimer[3].Q THEN
       #statMBMasterBuffer[2].MB_ADDR := 2;
       #statMBMasterBuffer[2].MODE := #Mode_Read;
       #statMBMasterBuffer[2].DATA_ADDR := #Addr_TempPV;
       #statMBMasterBuffer[2].DATA_LEN := 4;
   END_IF;
   #"statE5CC[2]".statReadReq[0] := #statTimer[3].Q;
   #_w1 := #statTimer[3].Q AND #statMBMasterBuffer[2].DONE AND NOT #statPulse[2];   // rising edge of #statMBMasterBuffer[2].DONE
   #statPulse[2] := #statMBMasterBuffer[2].DONE;
   IF #_w1 THEN
       #"statE5CC[2]".statReadTempPV := DINT_TO_REAL(#statMBMasterBuffer[2].DataPTR[1]);
       #"statE5CC[2]".statReadStatus := #statMBMasterBuffer[2].DataPTR[3];
       #"statE5CC[2]".statReadStep := 2;
   END_IF;
END_REGION

REGION Network 24: E5CC[2] -Read TempSP + AlarmValue1 ~ AlarmValue2_LowerLimit Commad
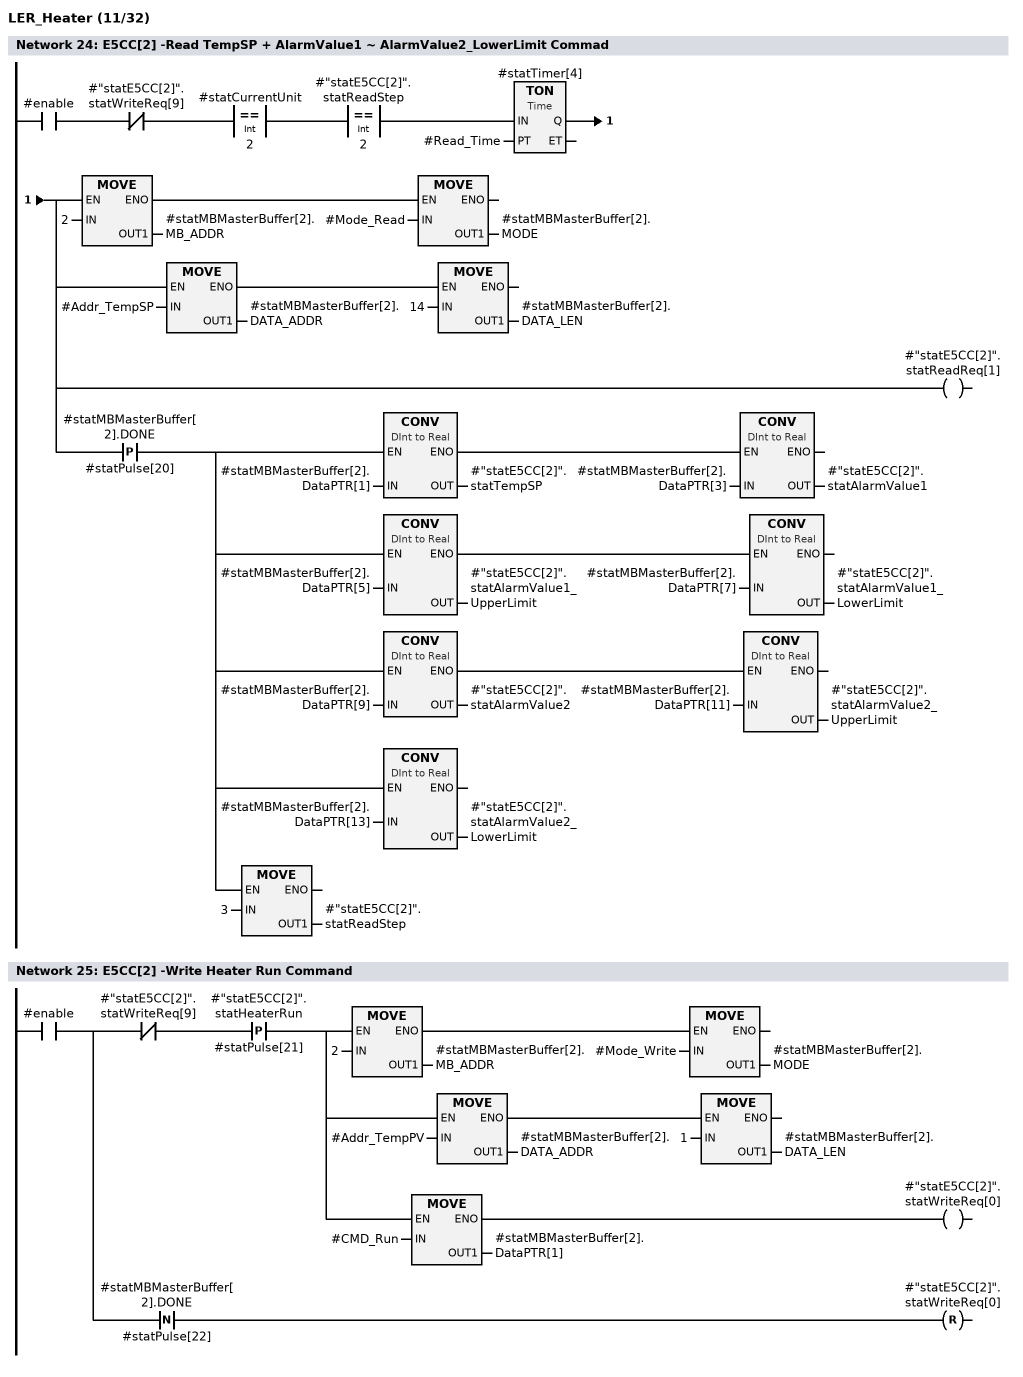
   RUNG wire#powerrail
      Contact( #enable )
      I_Contact( #"statE5CC[2]".statWriteReq[9] )
      { S7_Templates := "SrcType := Int" } EQ_Contact(in1 := #statCurrentUnit, in2 := 2)
      { S7_Templates := "SrcType := Int" } EQ_Contact(in1 := #"statE5CC[2]".statReadStep, in2 := 2)
      { S7_Templates := "time_type := Time" } #statTimer[4].TON(pt := #Read_Time, et =>)
      wire#w1
      Move(in := 2, out1 => #statMBMasterBuffer[2].MB_ADDR)
      Move(in := #Mode_Read, out1 => #statMBMasterBuffer[2].MODE)
   END_RUNG
   RUNG wire#w1
      Move(in := #Addr_TempSP, out1 => #statMBMasterBuffer[2].DATA_ADDR)
      Move(in := 14, out1 => #statMBMasterBuffer[2].DATA_LEN)
   END_RUNG
   RUNG wire#w1
      Coil( #"statE5CC[2]".statReadReq[1] )
   END_RUNG
   RUNG wire#w1
      P_Contact(operand := #statMBMasterBuffer[2].DONE, bit := #statPulse[20])
      wire#w2
      { S7_Templates := "[SrcType := DInt, DestType := Real]" } Convert(in := #statMBMasterBuffer[2].DataPTR[1], out => #"statE5CC[2]".statTempSP)
      { S7_Templates := "[SrcType := DInt, DestType := Real]" } Convert(in := #statMBMasterBuffer[2].DataPTR[3], out => #"statE5CC[2]".statAlarmValue1)
   END_RUNG
   RUNG wire#w2
      { S7_Templates := "[SrcType := DInt, DestType := Real]" } Convert(in := #statMBMasterBuffer[2].DataPTR[5], out => #"statE5CC[2]".statAlarmValue1_UpperLimit)
      { S7_Templates := "[SrcType := DInt, DestType := Real]" } Convert(in := #statMBMasterBuffer[2].DataPTR[7], out => #"statE5CC[2]".statAlarmValue1_LowerLimit)
   END_RUNG
   RUNG wire#w2
      { S7_Templates := "[SrcType := DInt, DestType := Real]" } Convert(in := #statMBMasterBuffer[2].DataPTR[9], out => #"statE5CC[2]".statAlarmValue2)
      { S7_Templates := "[SrcType := DInt, DestType := Real]" } Convert(in := #statMBMasterBuffer[2].DataPTR[11], out => #"statE5CC[2]".statAlarmValue2_UpperLimit)
   END_RUNG
   RUNG wire#w2
      { S7_Templates := "[SrcType := DInt, DestType := Real]" } Convert(in := #statMBMasterBuffer[2].DataPTR[13], out => #"statE5CC[2]".statAlarmValue2_LowerLimit)
   END_RUNG
   RUNG wire#w2
      Move(in := 3, out1 => #"statE5CC[2]".statReadStep)
   END_RUNG
   // the same network as SCL:
   #statTimer[4].TON(IN := #enable AND NOT #"statE5CC[2]".statWriteReq[9] AND (#statCurrentUnit = 2) AND (#"statE5CC[2]".statReadStep = 2),
                     PT := #Read_Time);
   IF #statTimer[4].Q THEN
       #statMBMasterBuffer[2].MB_ADDR := 2;
       #statMBMasterBuffer[2].MODE := #Mode_Read;
       #statMBMasterBuffer[2].DATA_ADDR := #Addr_TempSP;
       #statMBMasterBuffer[2].DATA_LEN := 14;
   END_IF;
   #"statE5CC[2]".statReadReq[1] := #statTimer[4].Q;
   #_w1 := #statTimer[4].Q AND #statMBMasterBuffer[2].DONE AND NOT #statPulse[20];   // rising edge of #statMBMasterBuffer[2].DONE
   #statPulse[20] := #statMBMasterBuffer[2].DONE;
   IF #_w1 THEN
       #"statE5CC[2]".statTempSP := DINT_TO_REAL(#statMBMasterBuffer[2].DataPTR[1]);
       #"statE5CC[2]".statAlarmValue1 := DINT_TO_REAL(#statMBMasterBuffer[2].DataPTR[3]);
       #"statE5CC[2]".statAlarmValue1_UpperLimit := DINT_TO_REAL(#statMBMasterBuffer[2].DataPTR[5]);
       #"statE5CC[2]".statAlarmValue1_LowerLimit := DINT_TO_REAL(#statMBMasterBuffer[2].DataPTR[7]);
       #"statE5CC[2]".statAlarmValue2 := DINT_TO_REAL(#statMBMasterBuffer[2].DataPTR[9]);
       #"statE5CC[2]".statAlarmValue2_UpperLimit := DINT_TO_REAL(#statMBMasterBuffer[2].DataPTR[11]);
       #"statE5CC[2]".statAlarmValue2_LowerLimit := DINT_TO_REAL(#statMBMasterBuffer[2].DataPTR[13]);
       #"statE5CC[2]".statReadStep := 3;
   END_IF;
END_REGION

REGION Network 25: E5CC[2] -Write Heater Run Command
   RUNG wire#powerrail
      Contact( #enable )
      wire#w1
      I_Contact( #"statE5CC[2]".statWriteReq[9] )
      P_Contact(operand := #"statE5CC[2]".statHeaterRun, bit := #statPulse[21])
      wire#w2
      Move(in := 2, out1 => #statMBMasterBuffer[2].MB_ADDR)
      Move(in := #Mode_Write, out1 => #statMBMasterBuffer[2].MODE)
   END_RUNG
   RUNG wire#w2
      Move(in := #Addr_TempPV, out1 => #statMBMasterBuffer[2].DATA_ADDR)
      Move(in := 1, out1 => #statMBMasterBuffer[2].DATA_LEN)
   END_RUNG
   RUNG wire#w2
      Move(in := #CMD_Run, out1 => #statMBMasterBuffer[2].DataPTR[1])
      Coil( #"statE5CC[2]".statWriteReq[0] )
   END_RUNG
   RUNG wire#w1
      N_Contact(operand := #statMBMasterBuffer[2].DONE, bit := #statPulse[22])
      R_Coil( #"statE5CC[2]".statWriteReq[0] )
   END_RUNG
   // the same network as SCL:
   #_w1 := #enable AND NOT #"statE5CC[2]".statWriteReq[9] AND #"statE5CC[2]".statHeaterRun AND NOT #statPulse[21];   // rising edge of #"statE5CC[2]".statHeaterRun
   #statPulse[21] := #"statE5CC[2]".statHeaterRun;
   IF #_w1 THEN
       #statMBMasterBuffer[2].MB_ADDR := 2;
       #statMBMasterBuffer[2].MODE := #Mode_Write;
       #statMBMasterBuffer[2].DATA_ADDR := #Addr_TempPV;
       #statMBMasterBuffer[2].DATA_LEN := 1;
       #statMBMasterBuffer[2].DataPTR[1] := #CMD_Run;
   END_IF;
   #"statE5CC[2]".statWriteReq[0] := #_w1;
   #_w2 := #enable AND NOT #statMBMasterBuffer[2].DONE AND #statPulse[22];   // falling edge of #statMBMasterBuffer[2].DONE
   #statPulse[22] := #statMBMasterBuffer[2].DONE;
   IF #_w2 THEN #"statE5CC[2]".statWriteReq[0] := FALSE; END_IF;
END_REGION

REGION Network 26: E5CC[2] -Write Heater Stop Command
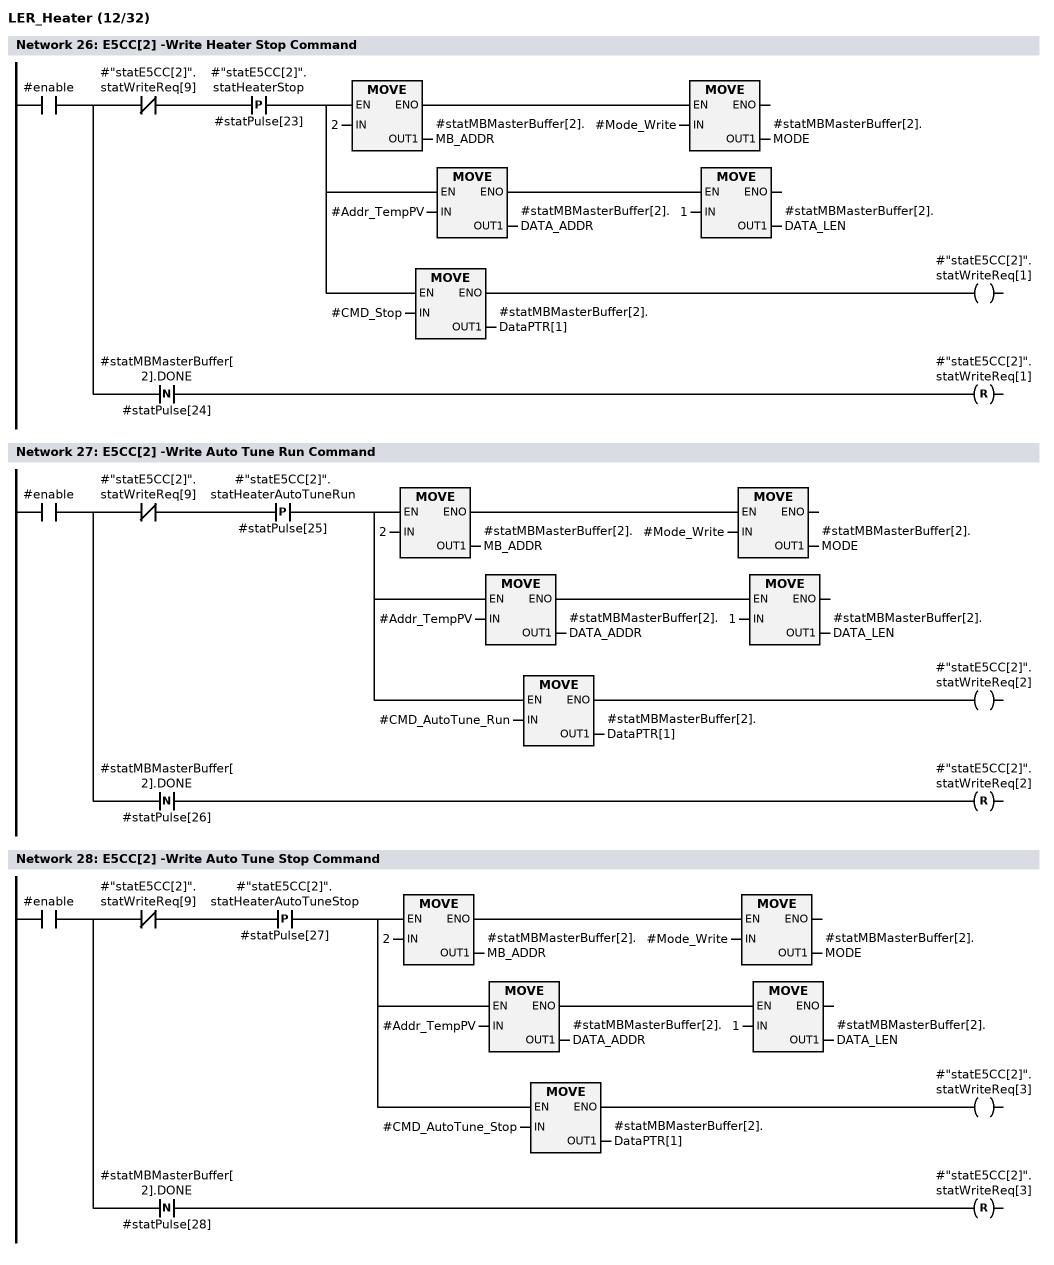
   RUNG wire#powerrail
      Contact( #enable )
      wire#w1
      I_Contact( #"statE5CC[2]".statWriteReq[9] )
      P_Contact(operand := #"statE5CC[2]".statHeaterStop, bit := #statPulse[23])
      wire#w2
      Move(in := 2, out1 => #statMBMasterBuffer[2].MB_ADDR)
      Move(in := #Mode_Write, out1 => #statMBMasterBuffer[2].MODE)
   END_RUNG
   RUNG wire#w2
      Move(in := #Addr_TempPV, out1 => #statMBMasterBuffer[2].DATA_ADDR)
      Move(in := 1, out1 => #statMBMasterBuffer[2].DATA_LEN)
   END_RUNG
   RUNG wire#w2
      Move(in := #CMD_Stop, out1 => #statMBMasterBuffer[2].DataPTR[1])
      Coil( #"statE5CC[2]".statWriteReq[1] )
   END_RUNG
   RUNG wire#w1
      N_Contact(operand := #statMBMasterBuffer[2].DONE, bit := #statPulse[24])
      R_Coil( #"statE5CC[2]".statWriteReq[1] )
   END_RUNG
   // the same network as SCL:
   #_w1 := #enable AND NOT #"statE5CC[2]".statWriteReq[9] AND #"statE5CC[2]".statHeaterStop AND NOT #statPulse[23];   // rising edge of #"statE5CC[2]".statHeaterStop
   #statPulse[23] := #"statE5CC[2]".statHeaterStop;
   IF #_w1 THEN
       #statMBMasterBuffer[2].MB_ADDR := 2;
       #statMBMasterBuffer[2].MODE := #Mode_Write;
       #statMBMasterBuffer[2].DATA_ADDR := #Addr_TempPV;
       #statMBMasterBuffer[2].DATA_LEN := 1;
       #statMBMasterBuffer[2].DataPTR[1] := #CMD_Stop;
   END_IF;
   #"statE5CC[2]".statWriteReq[1] := #_w1;
   #_w2 := #enable AND NOT #statMBMasterBuffer[2].DONE AND #statPulse[24];   // falling edge of #statMBMasterBuffer[2].DONE
   #statPulse[24] := #statMBMasterBuffer[2].DONE;
   IF #_w2 THEN #"statE5CC[2]".statWriteReq[1] := FALSE; END_IF;
END_REGION

REGION Network 27: E5CC[2] -Write Auto Tune Run Command
   RUNG wire#powerrail
      Contact( #enable )
      wire#w1
      I_Contact( #"statE5CC[2]".statWriteReq[9] )
      P_Contact(operand := #"statE5CC[2]".statHeaterAutoTuneRun, bit := #statPulse[25])
      wire#w2
      Move(in := 2, out1 => #statMBMasterBuffer[2].MB_ADDR)
      Move(in := #Mode_Write, out1 => #statMBMasterBuffer[2].MODE)
   END_RUNG
   RUNG wire#w2
      Move(in := #Addr_TempPV, out1 => #statMBMasterBuffer[2].DATA_ADDR)
      Move(in := 1, out1 => #statMBMasterBuffer[2].DATA_LEN)
   END_RUNG
   RUNG wire#w2
      Move(in := #CMD_AutoTune_Run, out1 => #statMBMasterBuffer[2].DataPTR[1])
      Coil( #"statE5CC[2]".statWriteReq[2] )
   END_RUNG
   RUNG wire#w1
      N_Contact(operand := #statMBMasterBuffer[2].DONE, bit := #statPulse[26])
      R_Coil( #"statE5CC[2]".statWriteReq[2] )
   END_RUNG
   // the same network as SCL:
   #_w1 := #enable AND NOT #"statE5CC[2]".statWriteReq[9] AND #"statE5CC[2]".statHeaterAutoTuneRun AND NOT #statPulse[25];   // rising edge of #"statE5CC[2]".statHeaterAutoTuneRun
   #statPulse[25] := #"statE5CC[2]".statHeaterAutoTuneRun;
   IF #_w1 THEN
       #statMBMasterBuffer[2].MB_ADDR := 2;
       #statMBMasterBuffer[2].MODE := #Mode_Write;
       #statMBMasterBuffer[2].DATA_ADDR := #Addr_TempPV;
       #statMBMasterBuffer[2].DATA_LEN := 1;
       #statMBMasterBuffer[2].DataPTR[1] := #CMD_AutoTune_Run;
   END_IF;
   #"statE5CC[2]".statWriteReq[2] := #_w1;
   #_w2 := #enable AND NOT #statMBMasterBuffer[2].DONE AND #statPulse[26];   // falling edge of #statMBMasterBuffer[2].DONE
   #statPulse[26] := #statMBMasterBuffer[2].DONE;
   IF #_w2 THEN #"statE5CC[2]".statWriteReq[2] := FALSE; END_IF;
END_REGION

REGION Network 28: E5CC[2] -Write Auto Tune Stop Command
   RUNG wire#powerrail
      Contact( #enable )
      wire#w1
      I_Contact( #"statE5CC[2]".statWriteReq[9] )
      P_Contact(operand := #"statE5CC[2]".statHeaterAutoTuneStop, bit := #statPulse[27])
      wire#w2
      Move(in := 2, out1 => #statMBMasterBuffer[2].MB_ADDR)
      Move(in := #Mode_Write, out1 => #statMBMasterBuffer[2].MODE)
   END_RUNG
   RUNG wire#w2
      Move(in := #Addr_TempPV, out1 => #statMBMasterBuffer[2].DATA_ADDR)
      Move(in := 1, out1 => #statMBMasterBuffer[2].DATA_LEN)
   END_RUNG
   RUNG wire#w2
      Move(in := #CMD_AutoTune_Stop, out1 => #statMBMasterBuffer[2].DataPTR[1])
      Coil( #"statE5CC[2]".statWriteReq[3] )
   END_RUNG
   RUNG wire#w1
      N_Contact(operand := #statMBMasterBuffer[2].DONE, bit := #statPulse[28])
      R_Coil( #"statE5CC[2]".statWriteReq[3] )
   END_RUNG
   // the same network as SCL:
   #_w1 := #enable AND NOT #"statE5CC[2]".statWriteReq[9] AND #"statE5CC[2]".statHeaterAutoTuneStop AND NOT #statPulse[27];   // rising edge of #"statE5CC[2]".statHeaterAutoTuneStop
   #statPulse[27] := #"statE5CC[2]".statHeaterAutoTuneStop;
   IF #_w1 THEN
       #statMBMasterBuffer[2].MB_ADDR := 2;
       #statMBMasterBuffer[2].MODE := #Mode_Write;
       #statMBMasterBuffer[2].DATA_ADDR := #Addr_TempPV;
       #statMBMasterBuffer[2].DATA_LEN := 1;
       #statMBMasterBuffer[2].DataPTR[1] := #CMD_AutoTune_Stop;
   END_IF;
   #"statE5CC[2]".statWriteReq[3] := #_w1;
   #_w2 := #enable AND NOT #statMBMasterBuffer[2].DONE AND #statPulse[28];   // falling edge of #statMBMasterBuffer[2].DONE
   #statPulse[28] := #statMBMasterBuffer[2].DONE;
   IF #_w2 THEN #"statE5CC[2]".statWriteReq[3] := FALSE; END_IF;
END_REGION

REGION Network 29: E5CC[2]-Write TempSP + AlarmValue1 ~ AlarmValue2_LowerLimit Command
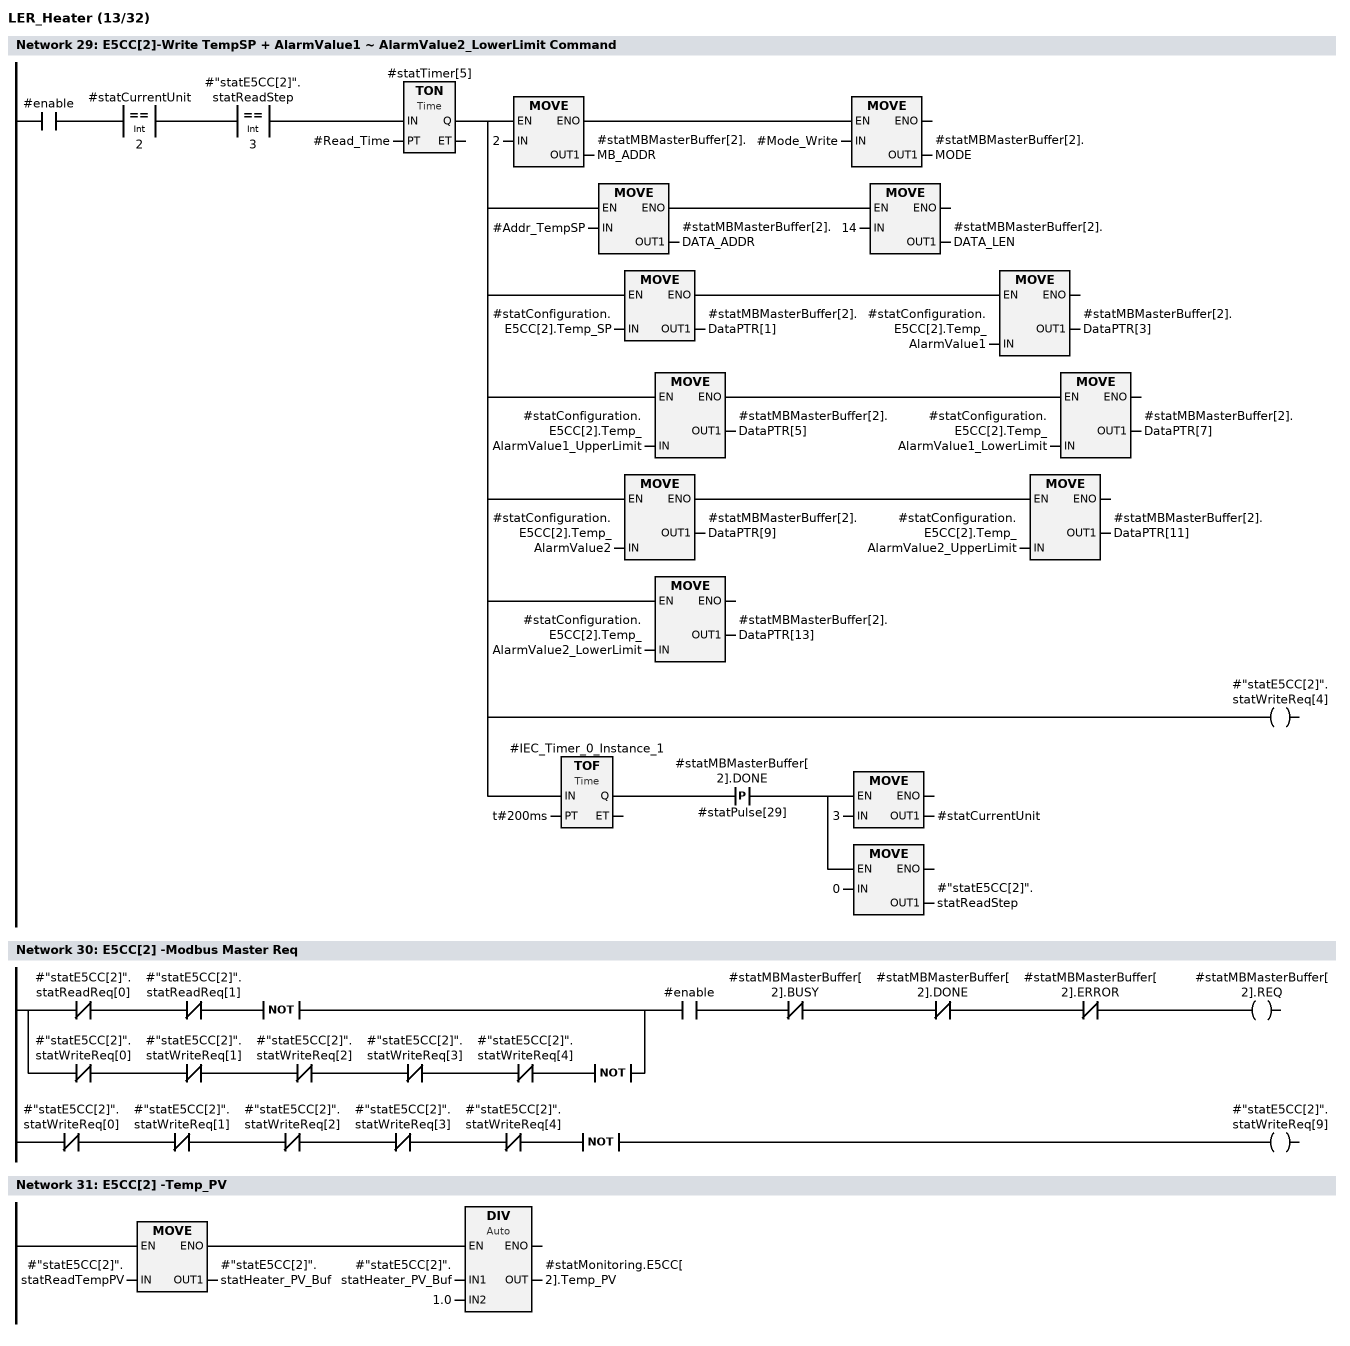
   RUNG wire#powerrail
      Contact( #enable )
      { S7_Templates := "SrcType := Int" } EQ_Contact(in1 := #statCurrentUnit, in2 := 2)
      { S7_Templates := "SrcType := Int" } EQ_Contact(in1 := #"statE5CC[2]".statReadStep, in2 := 3)
      { S7_Templates := "time_type := Time" } #statTimer[5].TON(pt := #Read_Time, et =>)
      wire#w1
      Move(in := 2, out1 => #statMBMasterBuffer[2].MB_ADDR)
      Move(in := #Mode_Write, out1 => #statMBMasterBuffer[2].MODE)
   END_RUNG
   RUNG wire#w1
      Move(in := #Addr_TempSP, out1 => #statMBMasterBuffer[2].DATA_ADDR)
      Move(in := 14, out1 => #statMBMasterBuffer[2].DATA_LEN)
   END_RUNG
   RUNG wire#w1
      Move(in := #statConfiguration.E5CC[2].Temp_SP, out1 => #statMBMasterBuffer[2].DataPTR[1])
      Move(in := #statConfiguration.E5CC[2].Temp_AlarmValue1, out1 => #statMBMasterBuffer[2].DataPTR[3])
   END_RUNG
   RUNG wire#w1
      Move(in := #statConfiguration.E5CC[2].Temp_AlarmValue1_UpperLimit, out1 => #statMBMasterBuffer[2].DataPTR[5])
      Move(in := #statConfiguration.E5CC[2].Temp_AlarmValue1_LowerLimit, out1 => #statMBMasterBuffer[2].DataPTR[7])
   END_RUNG
   RUNG wire#w1
      Move(in := #statConfiguration.E5CC[2].Temp_AlarmValue2, out1 => #statMBMasterBuffer[2].DataPTR[9])
      Move(in := #statConfiguration.E5CC[2].Temp_AlarmValue2_UpperLimit, out1 => #statMBMasterBuffer[2].DataPTR[11])
   END_RUNG
   RUNG wire#w1
      Move(in := #statConfiguration.E5CC[2].Temp_AlarmValue2_LowerLimit, out1 => #statMBMasterBuffer[2].DataPTR[13])
   END_RUNG
   RUNG wire#w1
      Coil( #"statE5CC[2]".statWriteReq[4] )
   END_RUNG
   RUNG wire#w1
      { S7_Templates := "time_type := Time" } #IEC_Timer_0_Instance_1.TOF(pt := t#200ms, et =>)
      P_Contact(operand := #statMBMasterBuffer[2].DONE, bit := #statPulse[29])
      wire#w2
      Move(in := 3, out1 => #statCurrentUnit)
   END_RUNG
   RUNG wire#w2
      Move(in := 0, out1 => #"statE5CC[2]".statReadStep)
   END_RUNG
   // the same network as SCL:
   #statTimer[5].TON(IN := #enable AND (#statCurrentUnit = 2) AND (#"statE5CC[2]".statReadStep = 3),
                     PT := #Read_Time);
   IF #statTimer[5].Q THEN
       #statMBMasterBuffer[2].MB_ADDR := 2;
       #statMBMasterBuffer[2].MODE := #Mode_Write;
       #statMBMasterBuffer[2].DATA_ADDR := #Addr_TempSP;
       #statMBMasterBuffer[2].DATA_LEN := 14;
       #statMBMasterBuffer[2].DataPTR[1] := #statConfiguration.E5CC[2].Temp_SP;
       #statMBMasterBuffer[2].DataPTR[3] := #statConfiguration.E5CC[2].Temp_AlarmValue1;
       #statMBMasterBuffer[2].DataPTR[5] := #statConfiguration.E5CC[2].Temp_AlarmValue1_UpperLimit;
       #statMBMasterBuffer[2].DataPTR[7] := #statConfiguration.E5CC[2].Temp_AlarmValue1_LowerLimit;
       #statMBMasterBuffer[2].DataPTR[9] := #statConfiguration.E5CC[2].Temp_AlarmValue2;
       #statMBMasterBuffer[2].DataPTR[11] := #statConfiguration.E5CC[2].Temp_AlarmValue2_UpperLimit;
       #statMBMasterBuffer[2].DataPTR[13] := #statConfiguration.E5CC[2].Temp_AlarmValue2_LowerLimit;
   END_IF;
   #"statE5CC[2]".statWriteReq[4] := #statTimer[5].Q;
   #IEC_Timer_0_Instance_1(IN := #statTimer[5].Q, PT := t#200ms);   // TOF
   #_w1 := #IEC_Timer_0_Instance_1.Q AND #statMBMasterBuffer[2].DONE AND NOT #statPulse[29];   // rising edge of #statMBMasterBuffer[2].DONE
   #statPulse[29] := #statMBMasterBuffer[2].DONE;
   IF #_w1 THEN
       #statCurrentUnit := 3;
       #"statE5CC[2]".statReadStep := 0;
   END_IF;
END_REGION

REGION Network 30: E5CC[2] -Modbus Master Req
   RUNG wire#powerrail
      I_Contact( #"statE5CC[2]".statReadReq[0] )
      I_Contact( #"statE5CC[2]".statReadReq[1] )
      Not()
      wire#w1
      Contact( #enable )
      I_Contact( #statMBMasterBuffer[2].BUSY )
      I_Contact( #statMBMasterBuffer[2].DONE )
      I_Contact( #statMBMasterBuffer[2].ERROR )
      Coil( #statMBMasterBuffer[2].REQ )
   END_RUNG
   RUNG wire#powerrail
      I_Contact( #"statE5CC[2]".statWriteReq[0] )
      I_Contact( #"statE5CC[2]".statWriteReq[1] )
      I_Contact( #"statE5CC[2]".statWriteReq[2] )
      I_Contact( #"statE5CC[2]".statWriteReq[3] )
      I_Contact( #"statE5CC[2]".statWriteReq[4] )
      Not()
   END_RUNG wire#w1
   RUNG wire#powerrail
      I_Contact( #"statE5CC[2]".statWriteReq[0] )
      I_Contact( #"statE5CC[2]".statWriteReq[1] )
      I_Contact( #"statE5CC[2]".statWriteReq[2] )
      I_Contact( #"statE5CC[2]".statWriteReq[3] )
      I_Contact( #"statE5CC[2]".statWriteReq[4] )
      Not()
      Coil( #"statE5CC[2]".statWriteReq[9] )
   END_RUNG
   // the same network as SCL:
   #statMBMasterBuffer[2].REQ := (NOT (NOT #"statE5CC[2]".statReadReq[0] AND NOT #"statE5CC[2]".statReadReq[1]) OR NOT (NOT #"statE5CC[2]".statWriteReq[0] AND NOT #"statE5CC[2]".statWriteReq[1] AND NOT #"statE5CC[2]".statWriteReq[2] AND NOT #"statE5CC[2]".statWriteReq[3] AND NOT #"statE5CC[2]".statWriteReq[4])) AND #enable AND NOT #statMBMasterBuffer[2].BUSY AND NOT #statMBMasterBuffer[2].DONE AND NOT #statMBMasterBuffer[2].ERROR;
   #"statE5CC[2]".statWriteReq[9] := NOT (NOT #"statE5CC[2]".statWriteReq[0] AND NOT #"statE5CC[2]".statWriteReq[1] AND NOT #"statE5CC[2]".statWriteReq[2] AND NOT #"statE5CC[2]".statWriteReq[3] AND NOT #"statE5CC[2]".statWriteReq[4]);
END_REGION

REGION Network 31: E5CC[2] -Temp_PV
   RUNG wire#powerrail
      Move(in := #"statE5CC[2]".statReadTempPV, out1 => #"statE5CC[2]".statHeater_PV_Buf)
      Div(in1 := #"statE5CC[2]".statHeater_PV_Buf, in2 := 1.0, out => #statMonitoring.E5CC[2].Temp_PV)
   END_RUNG
   // the same network as SCL:
   #"statE5CC[2]".statHeater_PV_Buf := #"statE5CC[2]".statReadTempPV;
   #statMonitoring.E5CC[2].Temp_PV := #"statE5CC[2]".statHeater_PV_Buf / 1.0;
END_REGION

REGION Network 32: E5CC[2] -Temp_PV Complete Check
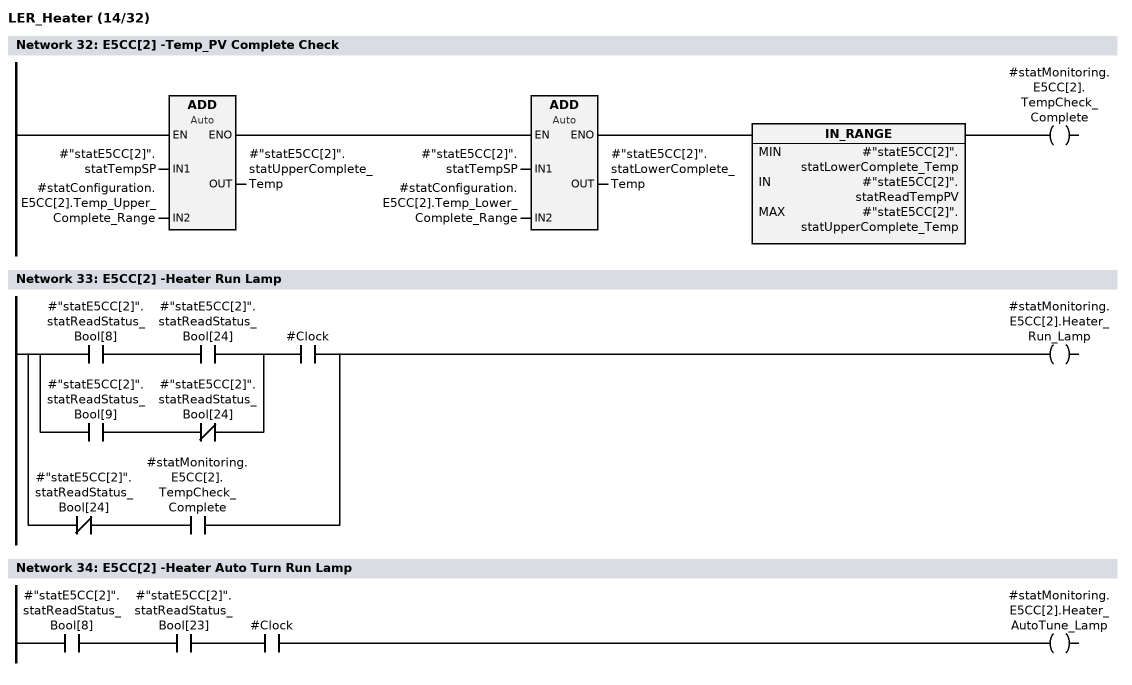
   RUNG wire#powerrail
      Add(in1 := #"statE5CC[2]".statTempSP, in2 := #statConfiguration.E5CC[2].Temp_Upper_Complete_Range, out => #"statE5CC[2]".statUpperComplete_Temp)
      Add(in1 := #"statE5CC[2]".statTempSP, in2 := #statConfiguration.E5CC[2].Temp_Lower_Complete_Range, out => #"statE5CC[2]".statLowerComplete_Temp)
      { S7_Templates := "SrcType := Real" } InRange(min := #"statE5CC[2]".statLowerComplete_Temp, in := #"statE5CC[2]".statReadTempPV, max := #"statE5CC[2]".statUpperComplete_Temp)
      Coil( #statMonitoring.E5CC[2].TempCheck_Complete )
   END_RUNG
   // the same network as SCL:
   #"statE5CC[2]".statUpperComplete_Temp := #"statE5CC[2]".statTempSP + #statConfiguration.E5CC[2].Temp_Upper_Complete_Range;
   #"statE5CC[2]".statLowerComplete_Temp := #"statE5CC[2]".statTempSP + #statConfiguration.E5CC[2].Temp_Lower_Complete_Range;
   #statMonitoring.E5CC[2].TempCheck_Complete := (#"statE5CC[2]".statLowerComplete_Temp <= #"statE5CC[2]".statReadTempPV) AND (#"statE5CC[2]".statReadTempPV <= #"statE5CC[2]".statUpperComplete_Temp);
END_REGION

REGION Network 33: E5CC[2] -Heater Run Lamp
   RUNG wire#powerrail
      Contact( #"statE5CC[2]".statReadStatus_Bool[8] )
      Contact( #"statE5CC[2]".statReadStatus_Bool[24] )
      wire#w1
      Contact( #Clock )
      wire#w2
      Coil( #statMonitoring.E5CC[2].Heater_Run_Lamp )
   END_RUNG
   RUNG wire#powerrail
      Contact( #"statE5CC[2]".statReadStatus_Bool[9] )
      I_Contact( #"statE5CC[2]".statReadStatus_Bool[24] )
   END_RUNG wire#w1
   RUNG wire#powerrail
      I_Contact( #"statE5CC[2]".statReadStatus_Bool[24] )
      Contact( #statMonitoring.E5CC[2].TempCheck_Complete )
   END_RUNG wire#w2
   // the same network as SCL:
   #statMonitoring.E5CC[2].Heater_Run_Lamp := (((#"statE5CC[2]".statReadStatus_Bool[8] AND #"statE5CC[2]".statReadStatus_Bool[24]) OR (#"statE5CC[2]".statReadStatus_Bool[9] AND NOT #"statE5CC[2]".statReadStatus_Bool[24])) AND #Clock) OR (NOT #"statE5CC[2]".statReadStatus_Bool[24] AND #statMonitoring.E5CC[2].TempCheck_Complete);
END_REGION

REGION Network 34: E5CC[2] -Heater Auto Turn Run Lamp
   RUNG wire#powerrail
      Contact( #"statE5CC[2]".statReadStatus_Bool[8] )
      Contact( #"statE5CC[2]".statReadStatus_Bool[23] )
      Contact( #Clock )
      Coil( #statMonitoring.E5CC[2].Heater_AutoTune_Lamp )
   END_RUNG
   // the same network as SCL:
   #statMonitoring.E5CC[2].Heater_AutoTune_Lamp := #"statE5CC[2]".statReadStatus_Bool[8] AND #"statE5CC[2]".statReadStatus_Bool[23] AND #Clock;
END_REGION

REGION Network 35 (SCL): E5CC[2] -Error Check
   REGION  E5CC Error Status
       // Dword to Bool
       SCATTER(IN := #"statE5CC[2]".statReadStatus,
               OUT => #"statE5CC[2]".statReadStatus_Bool);
   END_REGION


   REGION Error Code Search
       IF #"statE5CC[2]".statReadStatus <> 0 THEN
           CASE #"statE5CC[2]".statReadStatus OF
               #ERR_HEATER_CURRENT_VALUE_EXCEEDED_CT1:
                   #statMonitoring.E5CC[2].Status := #ERR_HEATER_CURRENT_VALUE_EXCEEDED_CT1;
               #ERR_HEATER_CURRENT_VALUE_HOLD_CT1:
                   #statMonitoring.E5CC[2].Status := #ERR_HEATER_CURRENT_VALUE_HOLD_CT1;
               #ERR_AD_CONVERTER_ABNORMALITY:
                   #statMonitoring.E5CC[2].Status := #ERR_AD_CONVERTER_ABNORMALITY;
               #ERR_HS_SSR_FAULT_ALERT_CT1:
                   #statMonitoring.E5CC[2].Status := #ERR_HS_SSR_FAULT_ALERT_CT1;
               #ERR_RSP_INPUT_ABNORMALITIES:
                   #statMonitoring.E5CC[2].Status := #ERR_RSP_INPUT_ABNORMALITIES;
               #ERR_MORE_THAN_INPUT:
                   #statMonitoring.E5CC[2].Status := #ERR_MORE_THAN_INPUT;
               #ERR_POTENTIOMETER_INPUT_ABNORMAL:
                   #statMonitoring.E5CC[2].Status := #ERR_POTENTIOMETER_INPUT_ABNORMAL;
               #ERR_CONTROL_OUTPUT_HEATED_OPEN_OUTPUT:
                   #statMonitoring.E5CC[2].Status := #ERR_CONTROL_OUTPUT_HEATED_OPEN_OUTPUT;
               #ERR_CONTROL_OUTPUT_COOL_CLOSE_OUTPUT:
                   #statMonitoring.E5CC[2].Status := #ERR_CONTROL_OUTPUT_COOL_CLOSE_OUTPUT;
               #ERR_HEATER_OPEN_CIRCUIT_HB_ALARM_CT1:
                   #statMonitoring.E5CC[2].Status := #ERR_HEATER_OPEN_CIRCUIT_HB_ALARM_CT1;
               #ERR_HEATER_OPEN_CIRCUIT_HB_ALARM_CT2:
                   #statMonitoring.E5CC[2].Status := #ERR_HEATER_OPEN_CIRCUIT_HB_ALARM_CT2;
               #ERR_ALERT_1:
                   #statMonitoring.E5CC[2].Status := #ERR_ALERT_1;
               #ERR_ALERT_2:
                   #statMonitoring.E5CC[2].Status := #ERR_ALERT_2;
               #ERR_ALERT_3:
                   #statMonitoring.E5CC[2].Status := #ERR_ALERT_3;
               #ERR_PROGRAM_END_OUTPUT:
                   #statMonitoring.E5CC[2].Status := #ERR_PROGRAM_END_OUTPUT;
               #ERR_EVENT_INPUT_1:
                   #statMonitoring.E5CC[2].Status := #ERR_EVENT_INPUT_1;
               #ERR_EVENT_INPUT_2:
                   #statMonitoring.E5CC[2].Status := #ERR_EVENT_INPUT_2;
               #ERR_EVENT_INPUT_3:
                   #statMonitoring.E5CC[2].Status := #ERR_EVENT_INPUT_3;
               #ERR_EVENT_INPUT_4:
                   #statMonitoring.E5CC[2].Status := #ERR_EVENT_INPUT_4;
               #ERR_WRITE_MODE:
                   #statMonitoring.E5CC[2].Status := #ERR_WRITE_MODE;
               #ERR_NON_VOLATILE_MEMORY:
                   #statMonitoring.E5CC[2].Status := #ERR_NON_VOLATILE_MEMORY;
               #ERR_SETTING_AREA:
                   #statMonitoring.E5CC[2].Status := #ERR_SETTING_AREA;
               #ERR_AT_RUN_STOP:
                   #statMonitoring.E5CC[2].Status := #ERR_AT_RUN_STOP;
               #ERR_RUN_STOP:
                   #statMonitoring.E5CC[2].Status := #ERR_RUN_STOP;
               #ERR_COMMUNICATION_WRITE:
                   #statMonitoring.E5CC[2].Status := #ERR_COMMUNICATION_WRITE;
               #ERR_AUTO_MANUAL:
                   #statMonitoring.E5CC[2].Status := #ERR_AUTO_MANUAL;
               #ERR_PROGRAM_START:
                   #statMonitoring.E5CC[2].Status := #ERR_PROGRAM_START;
               #ERR_HEATER_CURRENT_VALUE_EXCEEDED_CT2:
                   #statMonitoring.E5CC[2].Status := #ERR_HEATER_CURRENT_VALUE_EXCEEDED_CT2;
               #ERR_HEATER_CURRENT_VALUE_HOLD_CT2:
                   #statMonitoring.E5CC[2].Status := #ERR_HEATER_CURRENT_VALUE_HOLD_CT2;
               #ERR_HS_SSR_FAILURE_ALARM_CT2:
                   #statMonitoring.E5CC[2].Status := #ERR_HS_SSR_FAILURE_ALARM_CT2;
           END_CASE;
       ELSIF #"statE5CC[2]".statReadStatus = 0 THEN
           #statMonitoring.E5CC[2].Status := 0;
       END_IF;
   END_REGION

   #statMonitoring.E5CC[2].Error := #"statE5CC[2]".statReadStatus <> 0;
END_REGION

REGION Network 36 (SCL): E5CC[2] -##### Outputs mapping #####
   // Output Mapping
   #statMonitoring.E5CC[2].Temp_SP := #"statE5CC[2]".statTempSP;
   #statMonitoring.E5CC[2].Temp_AlarmValue1 := #"statE5CC[2]".statAlarmValue1;
   #statMonitoring.E5CC[2].Temp_AlarmValue1_UpperLimit := #"statE5CC[2]".statAlarmValue1_UpperLimit;
   #statMonitoring.E5CC[2].Temp_AlarmValue1_LowerLimit := #"statE5CC[2]".statAlarmValue1_LowerLimit;
   #statMonitoring.E5CC[2].Temp_AlarmValue2 := #"statE5CC[2]".statAlarmValue2;
   #statMonitoring.E5CC[2].Temp_AlarmValue2_UpperLimit := #"statE5CC[2]".statAlarmValue2_UpperLimit;
   #statMonitoring.E5CC[2].Temp_AlarmValue2_LowerLimit := #"statE5CC[2]".statAlarmValue2_LowerLimit;
   #statMonitoring.E5CC[2].E5CC_Status := #"statE5CC[2]".statReadStatus;
   #statMonitoring.E5CC[2].E5CC_Status_Bool := #"statE5CC[2]".statReadStatus_Bool;
END_REGION

REGION Network 37: E5CC[3] - ###### Input Mapping ######
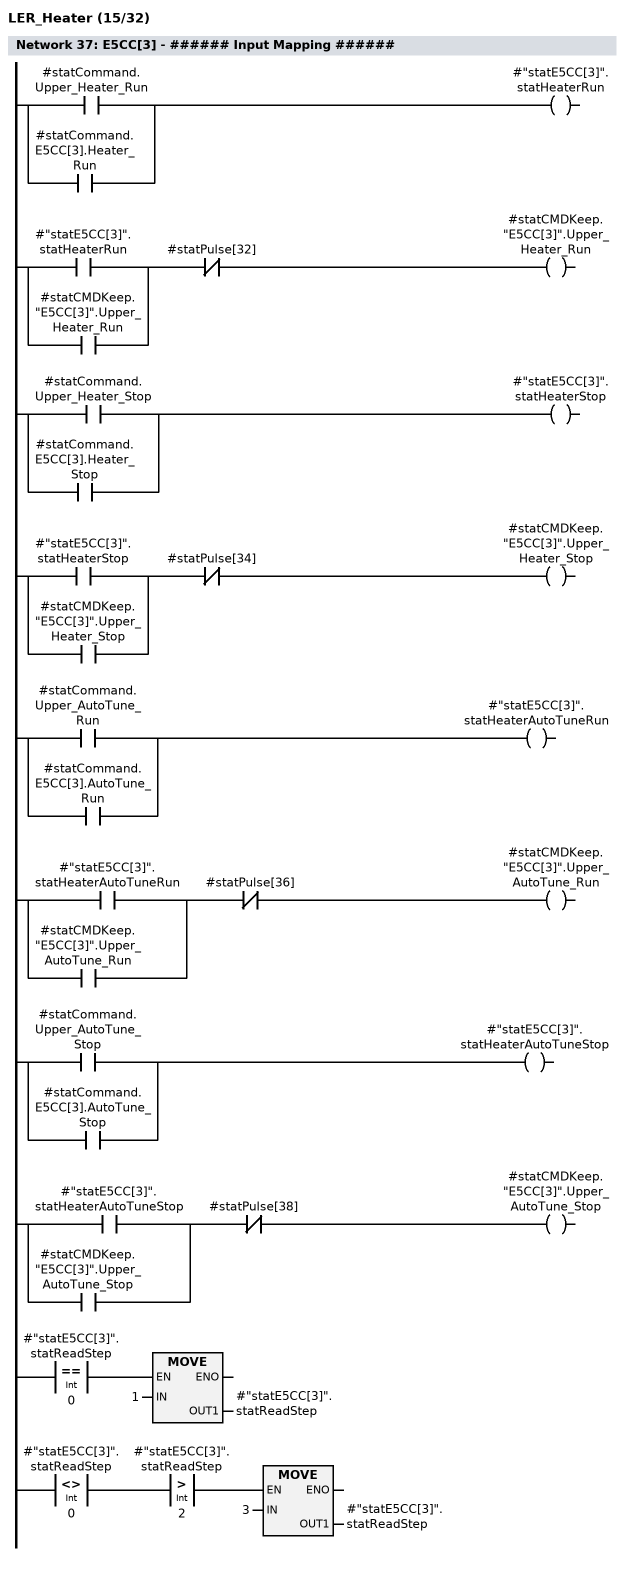
   RUNG wire#powerrail
      Contact( #statCommand.Upper_Heater_Run )
      wire#w1
      Coil( #"statE5CC[3]".statHeaterRun )
   END_RUNG
   RUNG wire#powerrail
      Contact( #statCommand.E5CC[3].Heater_Run )
   END_RUNG wire#w1
   RUNG wire#powerrail
      Contact( #"statE5CC[3]".statHeaterRun )
      wire#w2
      I_Contact( #statPulse[32] )
      Coil( #statCMDKeep."E5CC[3]".Upper_Heater_Run )
   END_RUNG
   RUNG wire#powerrail
      Contact( #statCMDKeep."E5CC[3]".Upper_Heater_Run )
   END_RUNG wire#w2
   RUNG wire#powerrail
      Contact( #statCommand.Upper_Heater_Stop )
      wire#w3
      Coil( #"statE5CC[3]".statHeaterStop )
   END_RUNG
   RUNG wire#powerrail
      Contact( #statCommand.E5CC[3].Heater_Stop )
   END_RUNG wire#w3
   RUNG wire#powerrail
      Contact( #"statE5CC[3]".statHeaterStop )
      wire#w4
      I_Contact( #statPulse[34] )
      Coil( #statCMDKeep."E5CC[3]".Upper_Heater_Stop )
   END_RUNG
   RUNG wire#powerrail
      Contact( #statCMDKeep."E5CC[3]".Upper_Heater_Stop )
   END_RUNG wire#w4
   RUNG wire#powerrail
      Contact( #statCommand.Upper_AutoTune_Run )
      wire#w5
      Coil( #"statE5CC[3]".statHeaterAutoTuneRun )
   END_RUNG
   RUNG wire#powerrail
      Contact( #statCommand.E5CC[3].AutoTune_Run )
   END_RUNG wire#w5
   RUNG wire#powerrail
      Contact( #"statE5CC[3]".statHeaterAutoTuneRun )
      wire#w6
      I_Contact( #statPulse[36] )
      Coil( #statCMDKeep."E5CC[3]".Upper_AutoTune_Run )
   END_RUNG
   RUNG wire#powerrail
      Contact( #statCMDKeep."E5CC[3]".Upper_AutoTune_Run )
   END_RUNG wire#w6
   RUNG wire#powerrail
      Contact( #statCommand.Upper_AutoTune_Stop )
      wire#w7
      Coil( #"statE5CC[3]".statHeaterAutoTuneStop )
   END_RUNG
   RUNG wire#powerrail
      Contact( #statCommand.E5CC[3].AutoTune_Stop )
   END_RUNG wire#w7
   RUNG wire#powerrail
      Contact( #"statE5CC[3]".statHeaterAutoTuneStop )
      wire#w8
      I_Contact( #statPulse[38] )
      Coil( #statCMDKeep."E5CC[3]".Upper_AutoTune_Stop )
   END_RUNG
   RUNG wire#powerrail
      Contact( #statCMDKeep."E5CC[3]".Upper_AutoTune_Stop )
   END_RUNG wire#w8
   RUNG wire#powerrail
      { S7_Templates := "SrcType := Int" } EQ_Contact(in1 := #"statE5CC[3]".statReadStep, in2 := 0)
      Move(in := 1, out1 => #"statE5CC[3]".statReadStep)
   END_RUNG
   RUNG wire#powerrail
      { S7_Templates := "SrcType := Int" } NE_Contact(in1 := #"statE5CC[3]".statReadStep, in2 := 0)
      { S7_Templates := "SrcType := Int" } GT_Contact(in1 := #"statE5CC[3]".statReadStep, in2 := 2)
      Move(in := 3, out1 => #"statE5CC[3]".statReadStep)
   END_RUNG
   // the same network as SCL:
   #"statE5CC[3]".statHeaterRun := #statCommand.Upper_Heater_Run OR #statCommand.E5CC[3].Heater_Run;
   #statCMDKeep."E5CC[3]".Upper_Heater_Run := (#"statE5CC[3]".statHeaterRun OR #statCMDKeep."E5CC[3]".Upper_Heater_Run) AND NOT #statPulse[32];
   #"statE5CC[3]".statHeaterStop := #statCommand.Upper_Heater_Stop OR #statCommand.E5CC[3].Heater_Stop;
   #statCMDKeep."E5CC[3]".Upper_Heater_Stop := (#"statE5CC[3]".statHeaterStop OR #statCMDKeep."E5CC[3]".Upper_Heater_Stop) AND NOT #statPulse[34];
   #"statE5CC[3]".statHeaterAutoTuneRun := #statCommand.Upper_AutoTune_Run OR #statCommand.E5CC[3].AutoTune_Run;
   #statCMDKeep."E5CC[3]".Upper_AutoTune_Run := (#"statE5CC[3]".statHeaterAutoTuneRun OR #statCMDKeep."E5CC[3]".Upper_AutoTune_Run) AND NOT #statPulse[36];
   #"statE5CC[3]".statHeaterAutoTuneStop := #statCommand.Upper_AutoTune_Stop OR #statCommand.E5CC[3].AutoTune_Stop;
   #statCMDKeep."E5CC[3]".Upper_AutoTune_Stop := (#"statE5CC[3]".statHeaterAutoTuneStop OR #statCMDKeep."E5CC[3]".Upper_AutoTune_Stop) AND NOT #statPulse[38];
   IF #"statE5CC[3]".statReadStep = 0 THEN #"statE5CC[3]".statReadStep := 1; END_IF;
   IF (#"statE5CC[3]".statReadStep <> 0) AND (#"statE5CC[3]".statReadStep > 2) THEN
       #"statE5CC[3]".statReadStep := 3;
   END_IF;
END_REGION

REGION Network 38: E5CC[3] -Read Temp PV + Status Command
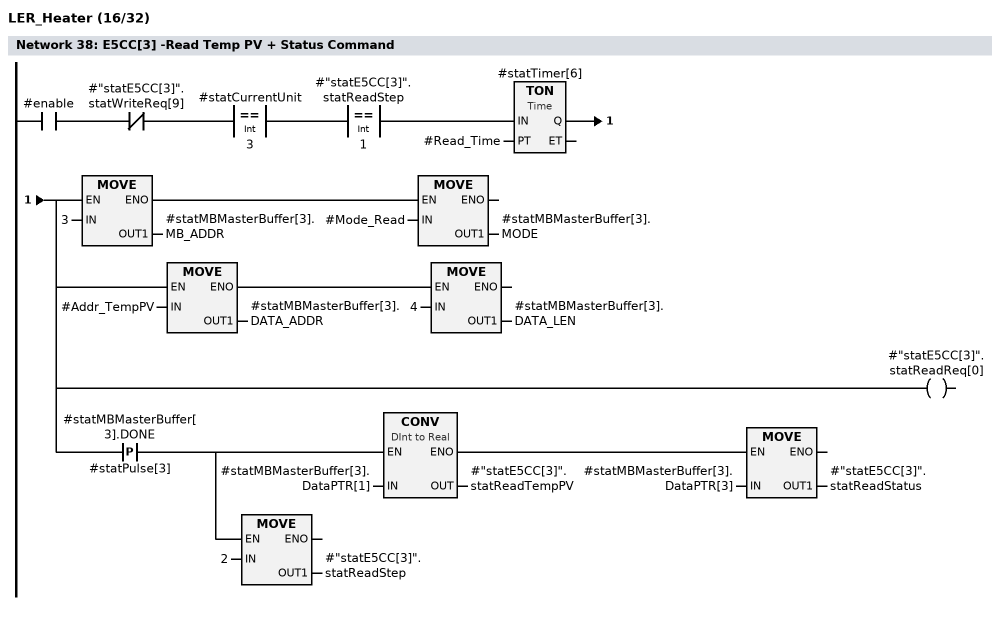
   RUNG wire#powerrail
      Contact( #enable )
      I_Contact( #"statE5CC[3]".statWriteReq[9] )
      { S7_Templates := "SrcType := Int" } EQ_Contact(in1 := #statCurrentUnit, in2 := 3)
      { S7_Templates := "SrcType := Int" } EQ_Contact(in1 := #"statE5CC[3]".statReadStep, in2 := 1)
      { S7_Templates := "time_type := Time" } #statTimer[6].TON(pt := #Read_Time, et =>)
      wire#w1
      Move(in := 3, out1 => #statMBMasterBuffer[3].MB_ADDR)
      Move(in := #Mode_Read, out1 => #statMBMasterBuffer[3].MODE)
   END_RUNG
   RUNG wire#w1
      Move(in := #Addr_TempPV, out1 => #statMBMasterBuffer[3].DATA_ADDR)
      Move(in := 4, out1 => #statMBMasterBuffer[3].DATA_LEN)
   END_RUNG
   RUNG wire#w1
      Coil( #"statE5CC[3]".statReadReq[0] )
   END_RUNG
   RUNG wire#w1
      P_Contact(operand := #statMBMasterBuffer[3].DONE, bit := #statPulse[3])
      wire#w2
      { S7_Templates := "[SrcType := DInt, DestType := Real]" } Convert(in := #statMBMasterBuffer[3].DataPTR[1], out => #"statE5CC[3]".statReadTempPV)
      Move(in := #statMBMasterBuffer[3].DataPTR[3], out1 => #"statE5CC[3]".statReadStatus)
   END_RUNG
   RUNG wire#w2
      Move(in := 2, out1 => #"statE5CC[3]".statReadStep)
   END_RUNG
   // the same network as SCL:
   #statTimer[6].TON(IN := #enable AND NOT #"statE5CC[3]".statWriteReq[9] AND (#statCurrentUnit = 3) AND (#"statE5CC[3]".statReadStep = 1),
                     PT := #Read_Time);
   IF #statTimer[6].Q THEN
       #statMBMasterBuffer[3].MB_ADDR := 3;
       #statMBMasterBuffer[3].MODE := #Mode_Read;
       #statMBMasterBuffer[3].DATA_ADDR := #Addr_TempPV;
       #statMBMasterBuffer[3].DATA_LEN := 4;
   END_IF;
   #"statE5CC[3]".statReadReq[0] := #statTimer[6].Q;
   #_w1 := #statTimer[6].Q AND #statMBMasterBuffer[3].DONE AND NOT #statPulse[3];   // rising edge of #statMBMasterBuffer[3].DONE
   #statPulse[3] := #statMBMasterBuffer[3].DONE;
   IF #_w1 THEN
       #"statE5CC[3]".statReadTempPV := DINT_TO_REAL(#statMBMasterBuffer[3].DataPTR[1]);
       #"statE5CC[3]".statReadStatus := #statMBMasterBuffer[3].DataPTR[3];
       #"statE5CC[3]".statReadStep := 2;
   END_IF;
END_REGION

REGION Network 39: E5CC[3] -Read TempSP + AlarmValue1 ~ AlarmValue2_LowerLimit Commad
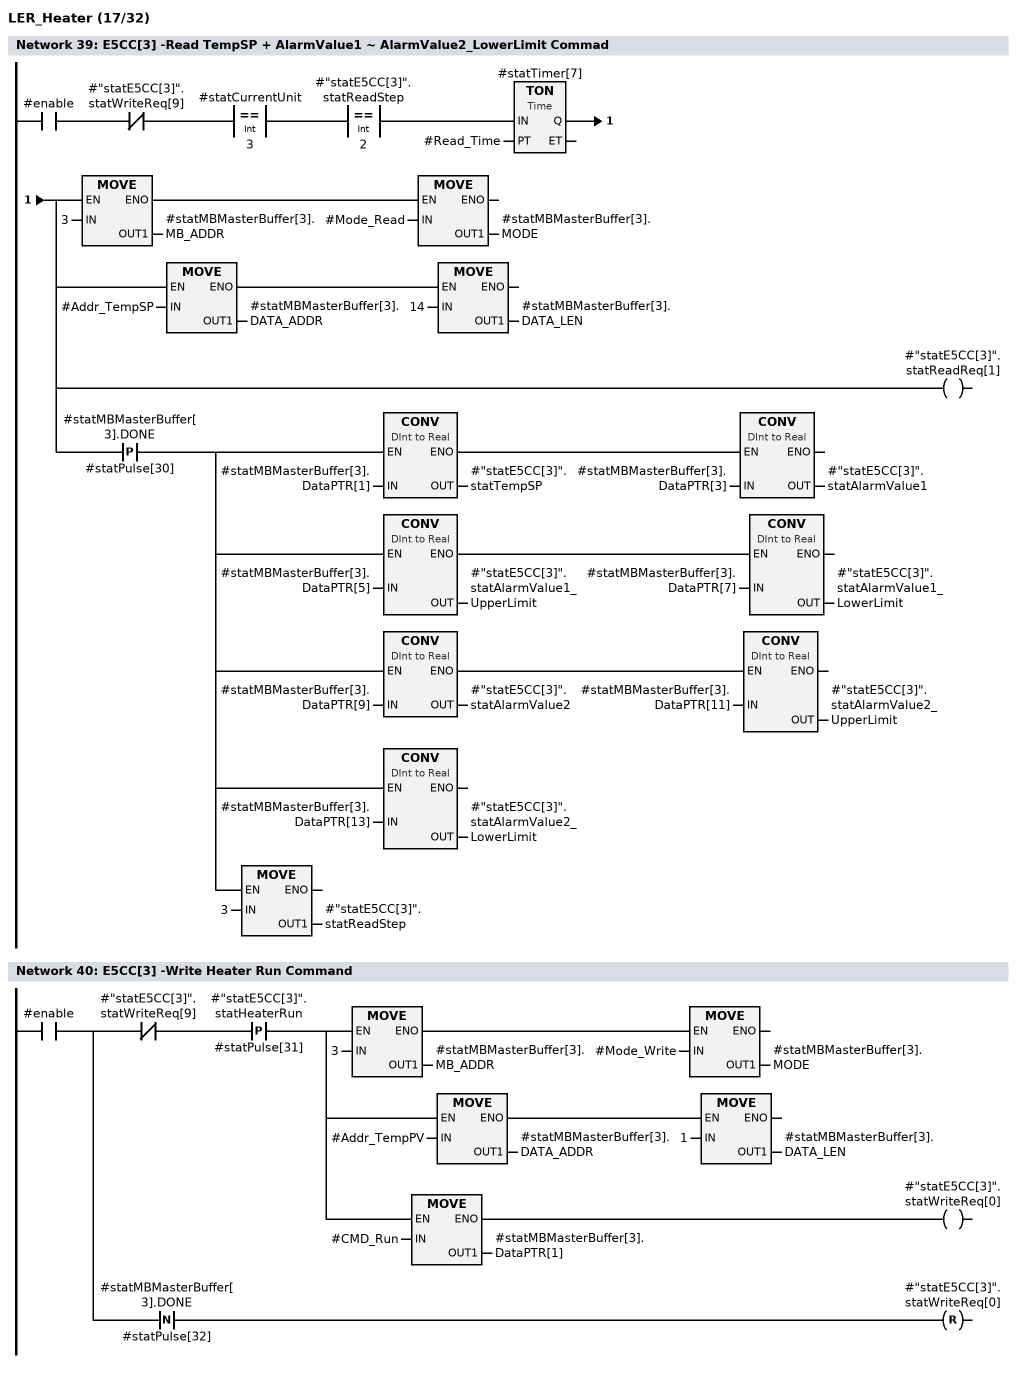
   RUNG wire#powerrail
      Contact( #enable )
      I_Contact( #"statE5CC[3]".statWriteReq[9] )
      { S7_Templates := "SrcType := Int" } EQ_Contact(in1 := #statCurrentUnit, in2 := 3)
      { S7_Templates := "SrcType := Int" } EQ_Contact(in1 := #"statE5CC[3]".statReadStep, in2 := 2)
      { S7_Templates := "time_type := Time" } #statTimer[7].TON(pt := #Read_Time, et =>)
      wire#w1
      Move(in := 3, out1 => #statMBMasterBuffer[3].MB_ADDR)
      Move(in := #Mode_Read, out1 => #statMBMasterBuffer[3].MODE)
   END_RUNG
   RUNG wire#w1
      Move(in := #Addr_TempSP, out1 => #statMBMasterBuffer[3].DATA_ADDR)
      Move(in := 14, out1 => #statMBMasterBuffer[3].DATA_LEN)
   END_RUNG
   RUNG wire#w1
      Coil( #"statE5CC[3]".statReadReq[1] )
   END_RUNG
   RUNG wire#w1
      P_Contact(operand := #statMBMasterBuffer[3].DONE, bit := #statPulse[30])
      wire#w2
      { S7_Templates := "[SrcType := DInt, DestType := Real]" } Convert(in := #statMBMasterBuffer[3].DataPTR[1], out => #"statE5CC[3]".statTempSP)
      { S7_Templates := "[SrcType := DInt, DestType := Real]" } Convert(in := #statMBMasterBuffer[3].DataPTR[3], out => #"statE5CC[3]".statAlarmValue1)
   END_RUNG
   RUNG wire#w2
      { S7_Templates := "[SrcType := DInt, DestType := Real]" } Convert(in := #statMBMasterBuffer[3].DataPTR[5], out => #"statE5CC[3]".statAlarmValue1_UpperLimit)
      { S7_Templates := "[SrcType := DInt, DestType := Real]" } Convert(in := #statMBMasterBuffer[3].DataPTR[7], out => #"statE5CC[3]".statAlarmValue1_LowerLimit)
   END_RUNG
   RUNG wire#w2
      { S7_Templates := "[SrcType := DInt, DestType := Real]" } Convert(in := #statMBMasterBuffer[3].DataPTR[9], out => #"statE5CC[3]".statAlarmValue2)
      { S7_Templates := "[SrcType := DInt, DestType := Real]" } Convert(in := #statMBMasterBuffer[3].DataPTR[11], out => #"statE5CC[3]".statAlarmValue2_UpperLimit)
   END_RUNG
   RUNG wire#w2
      { S7_Templates := "[SrcType := DInt, DestType := Real]" } Convert(in := #statMBMasterBuffer[3].DataPTR[13], out => #"statE5CC[3]".statAlarmValue2_LowerLimit)
   END_RUNG
   RUNG wire#w2
      Move(in := 3, out1 => #"statE5CC[3]".statReadStep)
   END_RUNG
   // the same network as SCL:
   #statTimer[7].TON(IN := #enable AND NOT #"statE5CC[3]".statWriteReq[9] AND (#statCurrentUnit = 3) AND (#"statE5CC[3]".statReadStep = 2),
                     PT := #Read_Time);
   IF #statTimer[7].Q THEN
       #statMBMasterBuffer[3].MB_ADDR := 3;
       #statMBMasterBuffer[3].MODE := #Mode_Read;
       #statMBMasterBuffer[3].DATA_ADDR := #Addr_TempSP;
       #statMBMasterBuffer[3].DATA_LEN := 14;
   END_IF;
   #"statE5CC[3]".statReadReq[1] := #statTimer[7].Q;
   #_w1 := #statTimer[7].Q AND #statMBMasterBuffer[3].DONE AND NOT #statPulse[30];   // rising edge of #statMBMasterBuffer[3].DONE
   #statPulse[30] := #statMBMasterBuffer[3].DONE;
   IF #_w1 THEN
       #"statE5CC[3]".statTempSP := DINT_TO_REAL(#statMBMasterBuffer[3].DataPTR[1]);
       #"statE5CC[3]".statAlarmValue1 := DINT_TO_REAL(#statMBMasterBuffer[3].DataPTR[3]);
       #"statE5CC[3]".statAlarmValue1_UpperLimit := DINT_TO_REAL(#statMBMasterBuffer[3].DataPTR[5]);
       #"statE5CC[3]".statAlarmValue1_LowerLimit := DINT_TO_REAL(#statMBMasterBuffer[3].DataPTR[7]);
       #"statE5CC[3]".statAlarmValue2 := DINT_TO_REAL(#statMBMasterBuffer[3].DataPTR[9]);
       #"statE5CC[3]".statAlarmValue2_UpperLimit := DINT_TO_REAL(#statMBMasterBuffer[3].DataPTR[11]);
       #"statE5CC[3]".statAlarmValue2_LowerLimit := DINT_TO_REAL(#statMBMasterBuffer[3].DataPTR[13]);
       #"statE5CC[3]".statReadStep := 3;
   END_IF;
END_REGION

REGION Network 40: E5CC[3] -Write Heater Run Command
   RUNG wire#powerrail
      Contact( #enable )
      wire#w1
      I_Contact( #"statE5CC[3]".statWriteReq[9] )
      P_Contact(operand := #"statE5CC[3]".statHeaterRun, bit := #statPulse[31])
      wire#w2
      Move(in := 3, out1 => #statMBMasterBuffer[3].MB_ADDR)
      Move(in := #Mode_Write, out1 => #statMBMasterBuffer[3].MODE)
   END_RUNG
   RUNG wire#w2
      Move(in := #Addr_TempPV, out1 => #statMBMasterBuffer[3].DATA_ADDR)
      Move(in := 1, out1 => #statMBMasterBuffer[3].DATA_LEN)
   END_RUNG
   RUNG wire#w2
      Move(in := #CMD_Run, out1 => #statMBMasterBuffer[3].DataPTR[1])
      Coil( #"statE5CC[3]".statWriteReq[0] )
   END_RUNG
   RUNG wire#w1
      N_Contact(operand := #statMBMasterBuffer[3].DONE, bit := #statPulse[32])
      R_Coil( #"statE5CC[3]".statWriteReq[0] )
   END_RUNG
   // the same network as SCL:
   #_w1 := #enable AND NOT #"statE5CC[3]".statWriteReq[9] AND #"statE5CC[3]".statHeaterRun AND NOT #statPulse[31];   // rising edge of #"statE5CC[3]".statHeaterRun
   #statPulse[31] := #"statE5CC[3]".statHeaterRun;
   IF #_w1 THEN
       #statMBMasterBuffer[3].MB_ADDR := 3;
       #statMBMasterBuffer[3].MODE := #Mode_Write;
       #statMBMasterBuffer[3].DATA_ADDR := #Addr_TempPV;
       #statMBMasterBuffer[3].DATA_LEN := 1;
       #statMBMasterBuffer[3].DataPTR[1] := #CMD_Run;
   END_IF;
   #"statE5CC[3]".statWriteReq[0] := #_w1;
   #_w2 := #enable AND NOT #statMBMasterBuffer[3].DONE AND #statPulse[32];   // falling edge of #statMBMasterBuffer[3].DONE
   #statPulse[32] := #statMBMasterBuffer[3].DONE;
   IF #_w2 THEN #"statE5CC[3]".statWriteReq[0] := FALSE; END_IF;
END_REGION

REGION Network 41: E5CC[3] -Write Heater Stop Command
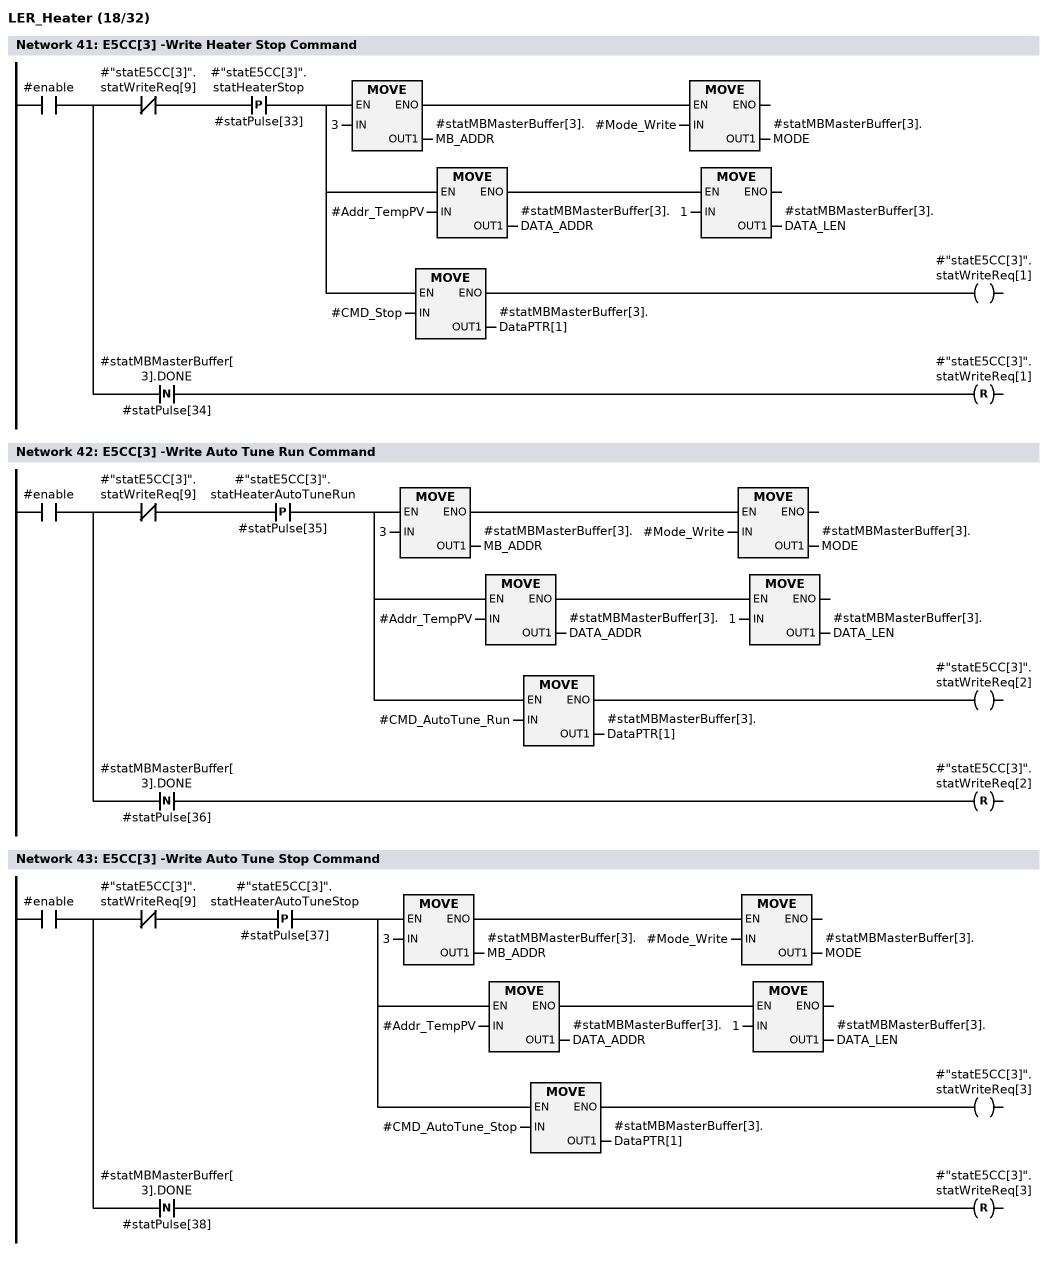
   RUNG wire#powerrail
      Contact( #enable )
      wire#w1
      I_Contact( #"statE5CC[3]".statWriteReq[9] )
      P_Contact(operand := #"statE5CC[3]".statHeaterStop, bit := #statPulse[33])
      wire#w2
      Move(in := 3, out1 => #statMBMasterBuffer[3].MB_ADDR)
      Move(in := #Mode_Write, out1 => #statMBMasterBuffer[3].MODE)
   END_RUNG
   RUNG wire#w2
      Move(in := #Addr_TempPV, out1 => #statMBMasterBuffer[3].DATA_ADDR)
      Move(in := 1, out1 => #statMBMasterBuffer[3].DATA_LEN)
   END_RUNG
   RUNG wire#w2
      Move(in := #CMD_Stop, out1 => #statMBMasterBuffer[3].DataPTR[1])
      Coil( #"statE5CC[3]".statWriteReq[1] )
   END_RUNG
   RUNG wire#w1
      N_Contact(operand := #statMBMasterBuffer[3].DONE, bit := #statPulse[34])
      R_Coil( #"statE5CC[3]".statWriteReq[1] )
   END_RUNG
   // the same network as SCL:
   #_w1 := #enable AND NOT #"statE5CC[3]".statWriteReq[9] AND #"statE5CC[3]".statHeaterStop AND NOT #statPulse[33];   // rising edge of #"statE5CC[3]".statHeaterStop
   #statPulse[33] := #"statE5CC[3]".statHeaterStop;
   IF #_w1 THEN
       #statMBMasterBuffer[3].MB_ADDR := 3;
       #statMBMasterBuffer[3].MODE := #Mode_Write;
       #statMBMasterBuffer[3].DATA_ADDR := #Addr_TempPV;
       #statMBMasterBuffer[3].DATA_LEN := 1;
       #statMBMasterBuffer[3].DataPTR[1] := #CMD_Stop;
   END_IF;
   #"statE5CC[3]".statWriteReq[1] := #_w1;
   #_w2 := #enable AND NOT #statMBMasterBuffer[3].DONE AND #statPulse[34];   // falling edge of #statMBMasterBuffer[3].DONE
   #statPulse[34] := #statMBMasterBuffer[3].DONE;
   IF #_w2 THEN #"statE5CC[3]".statWriteReq[1] := FALSE; END_IF;
END_REGION

REGION Network 42: E5CC[3] -Write Auto Tune Run Command
   RUNG wire#powerrail
      Contact( #enable )
      wire#w1
      I_Contact( #"statE5CC[3]".statWriteReq[9] )
      P_Contact(operand := #"statE5CC[3]".statHeaterAutoTuneRun, bit := #statPulse[35])
      wire#w2
      Move(in := 3, out1 => #statMBMasterBuffer[3].MB_ADDR)
      Move(in := #Mode_Write, out1 => #statMBMasterBuffer[3].MODE)
   END_RUNG
   RUNG wire#w2
      Move(in := #Addr_TempPV, out1 => #statMBMasterBuffer[3].DATA_ADDR)
      Move(in := 1, out1 => #statMBMasterBuffer[3].DATA_LEN)
   END_RUNG
   RUNG wire#w2
      Move(in := #CMD_AutoTune_Run, out1 => #statMBMasterBuffer[3].DataPTR[1])
      Coil( #"statE5CC[3]".statWriteReq[2] )
   END_RUNG
   RUNG wire#w1
      N_Contact(operand := #statMBMasterBuffer[3].DONE, bit := #statPulse[36])
      R_Coil( #"statE5CC[3]".statWriteReq[2] )
   END_RUNG
   // the same network as SCL:
   #_w1 := #enable AND NOT #"statE5CC[3]".statWriteReq[9] AND #"statE5CC[3]".statHeaterAutoTuneRun AND NOT #statPulse[35];   // rising edge of #"statE5CC[3]".statHeaterAutoTuneRun
   #statPulse[35] := #"statE5CC[3]".statHeaterAutoTuneRun;
   IF #_w1 THEN
       #statMBMasterBuffer[3].MB_ADDR := 3;
       #statMBMasterBuffer[3].MODE := #Mode_Write;
       #statMBMasterBuffer[3].DATA_ADDR := #Addr_TempPV;
       #statMBMasterBuffer[3].DATA_LEN := 1;
       #statMBMasterBuffer[3].DataPTR[1] := #CMD_AutoTune_Run;
   END_IF;
   #"statE5CC[3]".statWriteReq[2] := #_w1;
   #_w2 := #enable AND NOT #statMBMasterBuffer[3].DONE AND #statPulse[36];   // falling edge of #statMBMasterBuffer[3].DONE
   #statPulse[36] := #statMBMasterBuffer[3].DONE;
   IF #_w2 THEN #"statE5CC[3]".statWriteReq[2] := FALSE; END_IF;
END_REGION

REGION Network 43: E5CC[3] -Write Auto Tune Stop Command
   RUNG wire#powerrail
      Contact( #enable )
      wire#w1
      I_Contact( #"statE5CC[3]".statWriteReq[9] )
      P_Contact(operand := #"statE5CC[3]".statHeaterAutoTuneStop, bit := #statPulse[37])
      wire#w2
      Move(in := 3, out1 => #statMBMasterBuffer[3].MB_ADDR)
      Move(in := #Mode_Write, out1 => #statMBMasterBuffer[3].MODE)
   END_RUNG
   RUNG wire#w2
      Move(in := #Addr_TempPV, out1 => #statMBMasterBuffer[3].DATA_ADDR)
      Move(in := 1, out1 => #statMBMasterBuffer[3].DATA_LEN)
   END_RUNG
   RUNG wire#w2
      Move(in := #CMD_AutoTune_Stop, out1 => #statMBMasterBuffer[3].DataPTR[1])
      Coil( #"statE5CC[3]".statWriteReq[3] )
   END_RUNG
   RUNG wire#w1
      N_Contact(operand := #statMBMasterBuffer[3].DONE, bit := #statPulse[38])
      R_Coil( #"statE5CC[3]".statWriteReq[3] )
   END_RUNG
   // the same network as SCL:
   #_w1 := #enable AND NOT #"statE5CC[3]".statWriteReq[9] AND #"statE5CC[3]".statHeaterAutoTuneStop AND NOT #statPulse[37];   // rising edge of #"statE5CC[3]".statHeaterAutoTuneStop
   #statPulse[37] := #"statE5CC[3]".statHeaterAutoTuneStop;
   IF #_w1 THEN
       #statMBMasterBuffer[3].MB_ADDR := 3;
       #statMBMasterBuffer[3].MODE := #Mode_Write;
       #statMBMasterBuffer[3].DATA_ADDR := #Addr_TempPV;
       #statMBMasterBuffer[3].DATA_LEN := 1;
       #statMBMasterBuffer[3].DataPTR[1] := #CMD_AutoTune_Stop;
   END_IF;
   #"statE5CC[3]".statWriteReq[3] := #_w1;
   #_w2 := #enable AND NOT #statMBMasterBuffer[3].DONE AND #statPulse[38];   // falling edge of #statMBMasterBuffer[3].DONE
   #statPulse[38] := #statMBMasterBuffer[3].DONE;
   IF #_w2 THEN #"statE5CC[3]".statWriteReq[3] := FALSE; END_IF;
END_REGION

